# B&R Automation Studio project Agroittica
Automation Studio 4.9.5.36 SP; technology packages: mapp 5.18.0

## Configuration CP1382

CPU X20CP1382-RT, AutomationRuntime E4.83, Build 4.1.2, Safety 0.0, Vc V4.72.6

### Task classes (Cpu.sw)
```
Cyclic#1 (cycle 4000 us, tolerance 4000 us):
  Time <- main.Time.prg
  FIFO <- FIFO.FIFO.prg
  TCP_IP <- Tcp_ip.TCP_IP.prg
  Main <- main.Main.prg
  xsm_demo <- XSM_Demo_vnc.xsm_demo.prg
  xsm_demo_M <- XSM_Demo_vnc.xsm_demo_M2.prg
  Buffer_RPT <- main.Buffer_RPT.prg
  Laser_Enc <- IO.Laser_Enc.prg [disabled]
  Encoder <- IO.Encoder.prg [disabled]
Cyclic#2:
  Sim <- Sim.prg
Cyclic#3 (cycle 48000 us, tolerance 48000 us):
  RPT_CSV_ST <- main.RPT_CSV_ST.prg
Cyclic#4:
  Keys_Light <- Keys_Lights_combos.Keys_Lights.prg
  ip_adr <- XSM_Demo_vnc.ip_adr.prg  // Get ip address for VCN test.
  Recipe <- MpPkg.Recipe.prg
  Alarm_0 <- MpPkg.Alarm_0.prg
  Param_Fix <- main.Param_Fix.prg
  Hmi_Suppor <- Hmi.Hmi_Support.prg
  Login <- MpPkg.Login.prg [disabled]
DataObjects: Acp10sys
VcDataObjects: Visu_t <- Hmi.Visu_t30.dob, VGAvnc <- XSM_Demo_vnc.VGAvnc.dob, Visu <- Hmi.Visu.dob
Binaries: udbdef, arsvcreg, TCData, vcpdvnc, vcnet, vcbclass, vcrt, vcgclass, vccbtn, vcshared, vccline, vccnum, vcalarm, vccddbox, arialbd, vctcal, vcfntttf, vcdsloc, vcmgr, vccbmp, arial, vccpopup, vcpdsw, vcdsint, vcfile, vccovl, vccstr, vcctext, vccshape, vccdt, vccslider, vcchtml, vcclbox, vccscale, Visu_t01, Visu_t03, vcxml, Visu_t02, vccurl, vcpkat, vcchspot, vcpfar00, FWRules, vccalarm, Visu03, Visu01, Visu02, vcctrend, vccbar, vcpfx20, VGAvnc03, VGAvnc02, VGAvnc01, mvLoader, Acp10map, acp10cfg, ashwd, sysconf, asfw, arconfig, iomap, Recipes, AlarmHist, Alarm, ashwac, Config, Role, User, Config_1, VGAsvn01, VGAsvn03, VGAsvn02, visvc
Libraries: runtime, asstring, AsIOAcc, brsystem, AsMath, XSM_Ramp, AsIecCon, astime, Acp10_MC, sys_lib, Acp10man, Acp10par, NcGlobal, MpAlarmX, MpBase, MpRecipe, AsTCP, MpUser, MpFile, FileIO, dataobj, asarcfg, powerlnk, standard, vcresman, asbrstr, asusb, ashw, arssl, Library, visapi
```

### Hardware
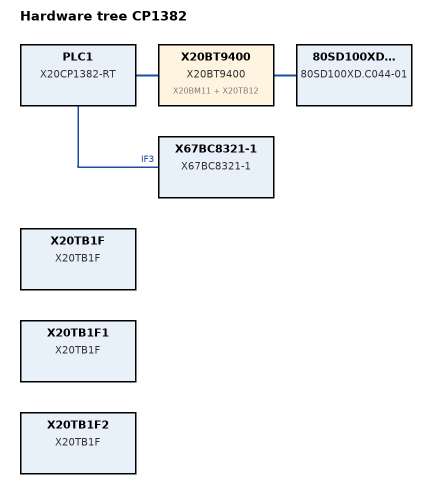
```
80SD100XD.C044-01 : 80SD100XD.C044-01 v2.2.0.0  [X2X1 -> X20BT9400.X2X1 [Cable Type=X2XCable, Length=10, Version=1.0.0.3]]
  FunctionModel = Ramp
  Supervision = off
  DirectionControl01 = on
PLC1 : X20CP1382-RT v1.11.0.0  [X1 -> X1.SL; X2 -> X2.SL; X3 -> X3.SL]
  Module X1 (Type=X1, Virtual=true, Version=1.11.0.0)
    Connection (Connector=SS1, TargetModule=X20TB1F, TargetConnector=SS)
    Connection (Connector=SL, TargetModule=PLC1, TargetConnector=X1)
    X1AI1_InputFilter = level 128
    X1AI1_InputLimitation = 4095
  Module X2 (Type=X2, Virtual=true, Version=1.11.0.0)
    Connection (Connector=SS1, TargetModule=X20TB1F1, TargetConnector=SS)
    Connection (Connector=SL, TargetModule=PLC1, TargetConnector=X2)
  Module X3 (Type=X3, Virtual=true, Version=1.11.0.0)
    Connection (Connector=SS1, TargetModule=X20TB1F2, TargetConnector=SS)
    Connection (Connector=SL, TargetModule=PLC1, TargetConnector=X3)
  Connector IF2:
    ActivateDevice = 1
    HostName = a07151
    Mode = Manual
    InternetAddress = 192.168.48.85
    SubnetMask = 255.255.255.0
    InaPort = 5555
    Vnc1
    VncVcObjectName1 = Visu_t
    VncKeyMappingFile1 = VC\PS2-Keyboard1.dis
    VncAuthentication1 = 1
    VncPasswordViewOnly1 = bazzica
    VncPasswordViewControl1 = promass
    VncMaxConnections1 = 10
    VncRefreshRate1 = 333
    Vnc2
    VncVcObjectName2 = VGAvnc
    VncKeyMappingFile2 = VC\PS2-Keyboard4.dis
    VncAuthentication2 = 1
    VncPasswordViewOnly2 = bazzica
    VncPasswordViewControl2 = promass
    VncPortNumber2 = 5901
    Vnc3
    VncVcObjectName3 = Visu
    VncKeyMappingFile3 = VC\PS2-Keyboard5.dis
    VncPortNumber3 = 5902
  Connector IF3:
    DNAConfiguration = manual
    CycleTime = 2000
    InaNodeNumber = 3
  ConfigurationID = Agroittica_CP1382
  RemanentGlobalPvSize = 100
  TimerDeviceType = EPLX2X
  TimerDevice = PLC1.IF3
  TaskClassIdleTime = 4000
  CyclicTaskClassCount = 4
  Cyclic1Duration = 4000
  Cyclic1Tolerance = 4000
  Cyclic3Duration = 48000
  Cyclic3Tolerance = 48000
  Cyclic8Duration = 8000
  FileDevice1
  FileDeviceName1 = Recipe
  FileDevicePath1 = C:\RECIPES
  FileDevice2
  FileDeviceName2 = Alarm
  FileDevicePath2 = C:\ALARM
  FileDevice3
  FileDeviceName3 = CF
  FileDevicePath3 = C:\
  FileDevice4
  FileDeviceName4 = DATA
  FileDevicePath4 = C:\DATA
  FileDevice5
  FileDeviceName5 = CFG
  FileDevicePath5 = C:\CFG
  FtpUser1
  FtpUsername1 = agroittica
  FtpUserPassword1 = lg+/2oVenYdo6VidhZ5rknSmVen51M+ANHGNxku/NAg=  // promass
  FtpUserSalt1 = EQR6eRm6
  FTPAccessRight1 = 0
  FTPdevice1 = ALL
  FtpUser2
  FtpUsername2 = bazzica
  FtpUserPassword2 = xgGZPKLqbdu5q4OkAcKaQyOUyno/5sjZu4T7S2DSwEQ=
  FtpUserSalt2 = nlL0YWjS
  FTPMSPartition2 = DATA
  ActivateOpcUa = 1
  OpcUaInformationModels_PV_Version = 1
  ReActionTaskDisabled = FALSE
X20BM11a : X20BM11 v1.0.0.1  [X2X1 -> PLC1.IF6]
X20BT9400 : X20BT9400 v1.1.0.0  [SS1 -> X20TB12a.SS; SL -> X20BM11a.SL1]
  Supervision = off
X20TB12a : X20TB12 v1.0.0.0
X20TB1F : X20TB1F v1.0.0.0
X20TB1F1 : X20TB1F v1.0.0.0
X20TB1F2 : X20TB1F v1.0.0.0
X67BC8321-1 : X67BC8321-1 v2.11.1.0  [PLK1 -> PLC1.IF3 (NodeNumber=3) [Cable Type=PowerlinkCable, Length=10, Version=1.0.0.3]]
  IOSupervision = off
  Direction01 = output
  Direction02 = output
  Direction03 = output
  Direction04 = output
  Direction05 = output
  Direction06 = output
```

### IoMap.iom - PLC1/IoMap.iom
```iecst
(********************************************************************
 * COPYRIGHT -- Bernecker + Rainer
 ********************************************************************
 * File: IoMap.iom
 * Author: leesa
 * Created: March 27, 2009
 ********************************************************************
 * IO mapping file
 ********************************************************************)
VAR_CONFIG
	::xsm_demo:XSM_Ctrl_0.IO_Mapping.ModuleOK AT %IX."80SD100XD.C044-01".ModuleOk;
	::xsm_demo:XSM_Ctrl_0.IO_Mapping.AbsPos AT %QD."80SD100XD.C044-01".AbsPos01;
	::xsm_demo:XSM_Ctrl_0.IO_Mapping.MpGenControl AT %QW."80SD100XD.C044-01".MpGenControl01;
	::xsm_demo:XSM_Ctrl_0.IO_Mapping.MpGenMode AT %QB."80SD100XD.C044-01".MpGenMode01;
	::xsm_demo:XSM_Ctrl_0.IO_Mapping.AbsPosActVal AT %ID."80SD100XD.C044-01".AbsPos01ActVal;
	::xsm_demo:XSM_Ctrl_0.IO_Mapping.MpGenStatus AT %IW."80SD100XD.C044-01".MpGenStatus01;
	::xsm_demo:XSM_Ctrl_0.IO_Mapping.InputStatus AT %IB."80SD100XD.C044-01".InputStatus;
	::xsm_demo:XSM_Ctrl_0.IO_Mapping.ModuleID AT %IW."80SD100XD.C044-01".ModuleID;
	glb_io.Di.Start AT %IX."X2".DigitalInput01;
	::xsm_demo:XSM_Ctrl_0.Enable AT %QX."X3".DigitalOutput01;
	glb_io.Do.Piston_gun_1 AT %QX."X3".DigitalOutput02;
	glb_io.Do.Piston_gun_2 AT %QX."X3".DigitalOutput04;
	Cyclic#1.Empty_Mag_22.Empty_Mag_Sensor AT %IX."X1".DigitalInput04;
	Cyclic#1.Empty_Mag_1_0.Empty_Mag_Sensor AT %IX."X1".DigitalInput02;
	::xsm_demo_M:XSM_Ctrl_2.IO_Mapping.AbsPos AT %QD."80SD100XD.C044-01".AbsPos02;
	::xsm_demo_M:XSM_Ctrl_2.IO_Mapping.MpGenControl AT %QW."80SD100XD.C044-01".MpGenControl02;
	::xsm_demo_M:XSM_Ctrl_2.IO_Mapping.MpGenMode AT %QB."80SD100XD.C044-01".MpGenMode02;
	::xsm_demo_M:XSM_Ctrl_2.IO_Mapping.AbsPosActVal AT %ID."80SD100XD.C044-01".AbsPos02ActVal;
	::xsm_demo_M:XSM_Ctrl_2.IO_Mapping.MpGenStatus AT %IW."80SD100XD.C044-01".MpGenStatus02;
	Cyclic#1.Feedback_0.Feedback_Em_Bt AT %IX."X2".DigitalInput13;
	Cyclic#1.Feedback_0.Feedback_Air AT %IX."X2".DigitalInput14;
	Cyclic#1.Beacon_1.Beeper_Alarm AT %QX."X67BC8321-1".IF1.ST1.DigitalOutput01;
	Cyclic#1.Beacon_2.Beeper_Alarm AT %QX."X67BC8321-1".IF1.ST1.DigitalOutput02;
	Cyclic#1.Beacon_1.White AT %QX."X67BC8321-1".IF1.ST1.DigitalOutput03;
	Cyclic#1.Beacon_2.White AT %QX."X67BC8321-1".IF1.ST1.DigitalOutput04;
	Cyclic#1.Beacon_1.Green AT %QX."X67BC8321-1".IF1.ST1.DigitalOutput05;
	Cyclic#1.Beacon_2.Green AT %QX."X67BC8321-1".IF1.ST1.DigitalOutput06;
	Cyclic#1.glb_io.Di.Si_03 AT %IX."X67BC8321-1".IF1.ST1.DigitalInput08;
	glb_io.Di.Powerlink AT %IX."X67BC8321-1".IF1.ST1.ModuleOk;
	glb_io.Do.Main_Piston_Up AT %QX."X3".DigitalOutput03;
	Cyclic#1.glb_io.Di.Si_01_raw AT %IX."X1".DigitalInput03;
	glb_io.Di.Automatic AT %IX."X2".DigitalInput02;
	glb_io.Di.Stop AT %IX."X2".DigitalInput03;
	glb_io.Di.Manual AT %IX."X2".DigitalInput04;
	glb_io.Di.Reset AT %IX."X2".DigitalInput05;
	glb_io.Di.Forward_Mag_1 AT %IX."X2".DigitalInput06;
	glb_io.Di.Forward_Mag_2 AT %IX."X2".DigitalInput07;
	glb_io.Di.Backward_Mag_1 AT %IX."X2".DigitalInput08;
	glb_io.Di.Backward_Mag_2 AT %IX."X2".DigitalInput09;
	glb_io.Do.Green_Light AT %QX."X3".DigitalOutput05;
	glb_io.Do.Red_Light AT %QX."X3".DigitalOutput06;
	glb_io.Do.Blue_Light AT %QX."X3".DigitalOutput07;
	glb_io.Do.Vacuum_On_Off AT %QX."X3".DigitalOutput08;
	Cyclic#1.::glb_io.Ai.Enc_laser_dist_raw AT %IW."X1".AnalogInput01;
	glb_io.Do.Main_Piston_Down AT %QX."X3".DigitalOutput09;
END_VAR
```

## Configuration CP1382_sim

### Task classes (Cpu.sw)
```
Cyclic#1 (cycle 4000 us, tolerance 4000 us):
  Sim <- Sim.prg
  Time <- main.Time.prg
  FIFO <- FIFO.FIFO.prg
  Main <- main.Main.prg
  xsm_demo <- XSM_Demo_vnc.xsm_demo.prg
  xsm_demo_M <- XSM_Demo_vnc.xsm_demo_M2.prg
  TCP_IP <- Tcp_ip.TCP_IP.prg
  Buffer_RPT <- main.Buffer_RPT.prg
  Laser_Enc <- IO.Laser_Enc.prg [disabled]
  Encoder <- IO.Encoder.prg [disabled]
Cyclic#3 (cycle 48000 us, tolerance 48000 us):
  RPT_CSV_ST <- main.RPT_CSV_ST.prg
Cyclic#4:
  Keys_Light <- Keys_Lights_combos.Keys_Lights.prg
  ip_adr <- XSM_Demo_vnc.ip_adr.prg  // Get ip address for VCN test.
  Recipe <- MpPkg.Recipe.prg
  Alarm_0 <- MpPkg.Alarm_0.prg
  Param_Fix <- main.Param_Fix.prg
  Hmi_Suppor <- Hmi.Hmi_Support.prg
  Login <- MpPkg.Login.prg [disabled]
DataObjects: Acp10sys
VcDataObjects: Visu_t <- Hmi.Visu_t30.dob, VGAvnc <- XSM_Demo_vnc.VGAvnc.dob, Visu <- Hmi.Visu.dob
Binaries: udbdef, arsvcreg, TCData, vcpdvnc, vcnet, vcbclass, vcrt, vcgclass, vccbtn, vcshared, vccline, vccnum, vcalarm, vccddbox, arialbd, vctcal, vcfntttf, vcdsloc, vcmgr, vccbmp, arial, vccpopup, vcpdsw, vcdsint, vcfile, vccovl, vccstr, vcctext, vccshape, vccdt, vccslider, vcchtml, vcclbox, vccscale, Visu_t01, Visu_t03, vcxml, Visu_t02, vccurl, vcpkat, vcchspot, vcpfar00, FWRules, vccalarm, Visu03, Visu01, Visu02, vcctrend, vccbar, VGAvnc03, VGAvnc02, VGAvnc01, mvLoader, Acp10map, acp10cfg, ashwd, sysconf, asfw, arconfig, iomap, Recipes, AlarmHist, Alarm, ashwac, Config, Role, User, Config_1, vcpfx20, VGAsvn01, VGAsvn03, VGAsvn02, visvc
ReActionTechnologyObjects: Program <- RT.Program.prg
Libraries: runtime, asstring, AsIOAcc, brsystem, AsMath, XSM_Ramp, AsIecCon, astime, Acp10_MC, sys_lib, Acp10man, Acp10par, NcGlobal, MpAlarmX, MpBase, MpRecipe, AsTCP, MpUser, MpFile, FileIO, dataobj, asarcfg, powerlnk, standard, vcresman, asbrstr, asusb, arssl, ashw, visapi, AsIORTI
```

### Hardware
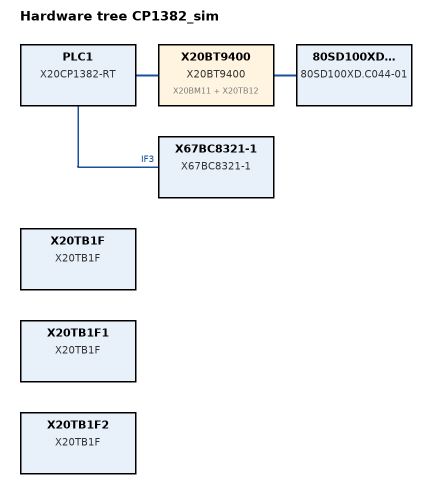
```
80SD100XD.C044-01 : 80SD100XD.C044-01 v2.2.0.0 (Disabled=true)  [X2X1 -> X20BT9400.X2X1 [Cable Type=X2XCable, Length=10, Version=1.0.0.3]]
  FunctionModel = Ramp
  Supervision = off
  DirectionControl01 = on
PLC1 : X20CP1382-RT v1.11.0.0  [X1 -> X1.SL; X2 -> X2.SL; X3 -> X3.SL]
  Module X1 (Type=X1, Virtual=true, Version=1.11.0.0)
    Connection (Connector=SS1, TargetModule=X20TB1F, TargetConnector=SS)
    Connection (Connector=SL, TargetModule=PLC1, TargetConnector=X1)
    X1AI1_InputFilter = level 128
    X1AI1_InputLimitation = 4095
  Module X2 (Type=X2, Virtual=true, Version=1.11.0.0)
    Connection (Connector=SS1, TargetModule=X20TB1F1, TargetConnector=SS)
    Connection (Connector=SL, TargetModule=PLC1, TargetConnector=X2)
  Module X3 (Type=X3, Virtual=true, Version=1.11.0.0)
    Connection (Connector=SS1, TargetModule=X20TB1F2, TargetConnector=SS)
    Connection (Connector=SL, TargetModule=PLC1, TargetConnector=X3)
  Connector IF2:
    ActivateDevice = 1
    HostName = a07151
    Mode = Manual
    InternetAddress = 192.168.48.85
    SubnetMask = 255.255.255.0
    InaPort = 5555
    Vnc1
    VncVcObjectName1 = Visu_t
    VncKeyMappingFile1 = VC\PS2-Keyboard1.dis
    VncAuthentication1 = 1
    VncPasswordViewOnly1 = bazzica
    VncPasswordViewControl1 = promass
    VncMaxConnections1 = 10
    VncRefreshRate1 = 333
    Vnc2
    VncVcObjectName2 = VGAvnc
    VncKeyMappingFile2 = VC\PS2-Keyboard4.dis
    VncAuthentication2 = 1
    VncPasswordViewOnly2 = bazzica
    VncPasswordViewControl2 = promass
    VncPortNumber2 = 5901
    Vnc3
    VncVcObjectName3 = Visu
    VncKeyMappingFile3 = VC\PS2-Keyboard5.dis
    VncPortNumber3 = 5902
  Connector IF3:
    DNAConfiguration = manual
    CycleTime = 2000
    InaNodeNumber = 3
  ConfigurationID = Agroittica_CP1382
  RemanentGlobalPvSize = 100
  TimerDeviceType = EPLX2X
  TimerDevice = PLC1.IF3
  TaskClassIdleTime = 4000
  CyclicTaskClassCount = 4
  Cyclic1Duration = 4000
  Cyclic1Tolerance = 4000
  Cyclic3Duration = 48000
  Cyclic3Tolerance = 48000
  Cyclic8Duration = 8000
  FileDevice1
  FileDeviceName1 = Recipe
  FileDevicePath1 = C:\RECIPES
  FileDevice2
  FileDeviceName2 = Alarm
  FileDevicePath2 = C:\ALARM
  FileDevice3
  FileDeviceName3 = CF
  FileDevicePath3 = C:\
  FileDevice4
  FileDeviceName4 = DATA
  FileDevicePath4 = C:\DATA
  FileDevice5
  FileDeviceName5 = CFG
  FileDevicePath5 = C:\CFG
  FtpUser1
  FtpUsername1 = agroittica
  FtpUserPassword1 = lg+/2oVenYdo6VidhZ5rknSmVen51M+ANHGNxku/NAg=  // promass
  FtpUserSalt1 = EQR6eRm6
  FTPAccessRight1 = 0
  FTPdevice1 = ALL
  FtpUser2
  FtpUsername2 = bazzica
  FtpUserPassword2 = xgGZPKLqbdu5q4OkAcKaQyOUyno/5sjZu4T7S2DSwEQ=
  FtpUserSalt2 = nlL0YWjS
  FTPMSPartition2 = DATA
  ActivateOpcUa = 1
  OpcUaInformationModels_PV_Version = 1
  ReActionTaskDisabled = FALSE
X20BM11a : X20BM11 v1.0.0.1 (Disabled=true)  [X2X1 -> PLC1.IF6]
X20BT9400 : X20BT9400 v1.1.0.0 (Disabled=true)  [SS1 -> X20TB12a.SS; SL -> X20BM11a.SL1]
  Supervision = off
X20TB12a : X20TB12 v1.0.0.0 (Disabled=true)
X20TB1F : X20TB1F v1.0.0.0
X20TB1F1 : X20TB1F v1.0.0.0
X20TB1F2 : X20TB1F v1.0.0.0
X67BC8321-1 : X67BC8321-1 v2.11.1.0 (Disabled=true)  [PLK1 -> PLC1.IF3 (NodeNumber=3) [Cable Type=PowerlinkCable, Length=10, Version=1.0.0.3]]
  Connector IF1 (Disabled=true)
  IOSupervision = off
  Direction01 = output
  Direction02 = output
  Direction03 = output
  Direction04 = output
  Direction05 = output
  Direction06 = output
```

### IoMap.iom - PLC1/IoMap.iom
```iecst
(********************************************************************
 * COPYRIGHT -- Bernecker + Rainer
 ********************************************************************
 * File: IoMap.iom
 * Author: leesa
 * Created: March 27, 2009
 ********************************************************************
 * IO mapping file
 ********************************************************************)
VAR_CONFIG
	::xsm_demo:XSM_Ctrl_0.IO_Mapping.ModuleOK AT %IX."80SD100XD.C044-01".ModuleOk;
	::xsm_demo:XSM_Ctrl_0.IO_Mapping.AbsPos AT %QD."80SD100XD.C044-01".AbsPos01;
	::xsm_demo:XSM_Ctrl_0.IO_Mapping.MpGenControl AT %QW."80SD100XD.C044-01".MpGenControl01;
	::xsm_demo:XSM_Ctrl_0.IO_Mapping.MpGenMode AT %QB."80SD100XD.C044-01".MpGenMode01;
	::xsm_demo:XSM_Ctrl_0.IO_Mapping.AbsPosActVal AT %ID."80SD100XD.C044-01".AbsPos01ActVal;
	::xsm_demo:XSM_Ctrl_0.IO_Mapping.MpGenStatus AT %IW."80SD100XD.C044-01".MpGenStatus01;
	::xsm_demo:XSM_Ctrl_0.IO_Mapping.InputStatus AT %IB."80SD100XD.C044-01".InputStatus;
	::xsm_demo:XSM_Ctrl_0.IO_Mapping.ModuleID AT %IW."80SD100XD.C044-01".ModuleID;
	glb_io.Di.Start AT %IX."X2".DigitalInput01;
	::xsm_demo:XSM_Ctrl_0.Enable AT %QX."X3".DigitalOutput01;
	glb_io.Do.Piston_gun_1 AT %QX."X3".DigitalOutput02;
	glb_io.Do.Piston_gun_2 AT %QX."X3".DigitalOutput04;
	Cyclic#1.Empty_Mag_22.Empty_Mag_Sensor AT %IX."X1".DigitalInput04;
	Cyclic#1.Empty_Mag_1_0.Empty_Mag_Sensor AT %IX."X1".DigitalInput02;
	::xsm_demo_M:XSM_Ctrl_2.IO_Mapping.AbsPos AT %QD."80SD100XD.C044-01".AbsPos02;
	::xsm_demo_M:XSM_Ctrl_2.IO_Mapping.MpGenControl AT %QW."80SD100XD.C044-01".MpGenControl02;
	::xsm_demo_M:XSM_Ctrl_2.IO_Mapping.MpGenMode AT %QB."80SD100XD.C044-01".MpGenMode02;
	::xsm_demo_M:XSM_Ctrl_2.IO_Mapping.AbsPosActVal AT %ID."80SD100XD.C044-01".AbsPos02ActVal;
	::xsm_demo_M:XSM_Ctrl_2.IO_Mapping.MpGenStatus AT %IW."80SD100XD.C044-01".MpGenStatus02;
	Cyclic#1.Feedback_0.Feedback_Em_Bt AT %IX."X2".DigitalInput13;
	Cyclic#1.Feedback_0.Feedback_Air AT %IX."X2".DigitalInput14;
	Cyclic#1.Beacon_1.Beeper_Alarm AT %QX."X67BC8321-1".IF1.ST1.DigitalOutput01;
	Cyclic#1.Beacon_2.Beeper_Alarm AT %QX."X67BC8321-1".IF1.ST1.DigitalOutput02;
	Cyclic#1.Beacon_1.White AT %QX."X67BC8321-1".IF1.ST1.DigitalOutput03;
	Cyclic#1.Beacon_2.White AT %QX."X67BC8321-1".IF1.ST1.DigitalOutput04;
	Cyclic#1.Beacon_1.Green AT %QX."X67BC8321-1".IF1.ST1.DigitalOutput05;
	Cyclic#1.Beacon_2.Green AT %QX."X67BC8321-1".IF1.ST1.DigitalOutput06;
	Cyclic#1.glb_io.Di.Si_03 AT %IX."X67BC8321-1".IF1.ST1.DigitalInput08;
	glb_io.Di.Powerlink AT %IX."X67BC8321-1".IF1.ST1.ModuleOk;
	glb_io.Do.Main_Piston_Up AT %QX."X3".DigitalOutput03;
	glb_io.Di.Si_01 AT %IX."X1".DigitalInput03;
	glb_io.Di.Automatic AT %IX."X2".DigitalInput02;
	glb_io.Di.Stop AT %IX."X2".DigitalInput03;
	glb_io.Di.Manual AT %IX."X2".DigitalInput04;
	glb_io.Di.Reset AT %IX."X2".DigitalInput05;
	glb_io.Di.Forward_Mag_1 AT %IX."X2".DigitalInput06;
	glb_io.Di.Backward_Mag_1 AT %IX."X2".DigitalInput08;
	glb_io.Di.Backward_Mag_2 AT %IX."X2".DigitalInput09;
	glb_io.Do.Green_Light AT %QX."X3".DigitalOutput05;
	glb_io.Do.Red_Light AT %QX."X3".DigitalOutput06;
	glb_io.Do.Blue_Light AT %QX."X3".DigitalOutput07;
	glb_io.Do.Vacuum_On_Off AT %QX."X3".DigitalOutput08;
	Cyclic#1.::glb_io.Ai.Enc_laser_dist_raw AT %IW."X1".AnalogInput01;
	glb_io.Do.Main_Piston_Down AT %QX."X3".DigitalOutput09;
	glb_io.Di.Forward_Mag_2 AT %IX."X2".DigitalInput07;
END_VAR
```

### Alarm.mpalarmxcore - PLC1/mappServices/Alarm.mpalarmxcore
```
Element gAlarmXCore (Type=mpalarmxcore)
  mapp.AlarmX.Core.Configuration:
    [0]:
      Name = Motor 1 fault
      Message = Motor 1 fault
      Behavior = PersistentAlarm
    [1]:
      Name = Air supply fault
      Message = Air supply not connected
      Behavior = PersistentAlarm
    [2]:
      Name = Emergency Button
      Message = Emergency Button
      Behavior = PersistentAlarm
    [3]:
      Name = Motor 2 fault
      Message = Motor 2 fault
      Behavior = PersistentAlarm
```

### Config.mpuser - PLC1/mappServices/Config.mpuser
```
Element UserMgmt (Type=mpuser)
  Groups:
    DefGroup#1:
      id = Admin
      level = 100
      admin = TRUE
      rights:
        [0] = FullAccess
        [1] = FullAccess
        [2] = FullAccess
        [3] = FullAccess
        [4] = FullAccess
    DefGroup#2:
      id = Operator
      rights:
        [0] = FullAccess
        [1] = StartOnly
        [2] = ViewOnly
        [3] = ViewOnly
        [4] = NoAccess
  Users:
    DefUser#1:
      id = Admin
      grp = Admin
      name = Default Admin User
      pwd = Admin
      pref = 
    DefUser#2:
      id = Operatore
      grp = Operator
      pwd = Agroittica
```

## Configuration CP1586

CPU X20CP1382-RT, AutomationRuntime E4.83, Build 4.1.2, Safety 0.0, Vc V4.72.6

### Task classes (Cpu.sw)
```
Cyclic#1:
  Main <- main.Main.prg
  Encoder <- IO.Encoder.prg
  xsm_demo <- XSM_Demo_vnc.xsm_demo.prg
Cyclic#4:
  ip_adr <- XSM_Demo_vnc.ip_adr.prg  // Get ip address for VCN test.
  Recipe <- MpPkg.Recipe.prg
  Alarm_0 <- MpPkg.Alarm_0.prg
  TCP_IP <- Tcp_ip.TCP_IP.prg
DataObjects: Acp10sys
VcDataObjects: VGAvnc <- XSM_Demo_vnc.VGAvnc.dob, Visu_t <- Hmi.Visu_t30.dob
Binaries: VGAvnc03, VGAvnc02, VGAvnc01, vcpdvnc, vcnet, vcbclass, vcrt, vcgclass, vccbtn, vcshared, vccline, vccnum, vcalarm, vccddbox, arialbd, vctcal, vcfntttf, vcdsloc, vcmgr, vccbmp, arial, vccpopup, vcpdsw, vcdsint, vcfile, vccovl, vccstr, vcctext, vccshape, vccdt, vccslider, vcchtml, vcclbox, vccscale, Visu_t01, Visu_t03, vcxml, Visu_t02, vccurl, vcpkat, udbdef, arsvcreg, vcchspot, TCData, vcpfx20, Acp10map, acp10cfg, ashwd, sysconf, asfw, arconfig, iomap, Recipes, AlarmHist, Alarm, ashwac, vcpfar00, VGAsvn01, VGAsvn03, VGAsvn02, visvc
Libraries: runtime, asstring, AsIOAcc, brsystem, AsMath, XSM_Ramp, AsIecCon, astime, Acp10_MC, sys_lib, Acp10man, Acp10par, NcGlobal, MpAlarmX, MpBase, MpRecipe, AsTCP, MpUser, vcresman, dataobj, asarcfg, fileio, powerlnk, standard, ashw, Library, visapi
```

### Hardware
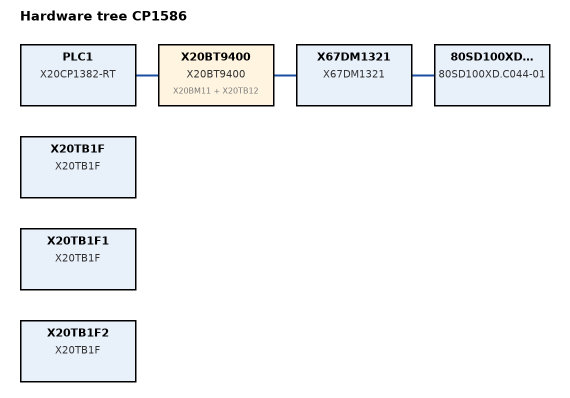
```
80SD100XD.C044-01 : 80SD100XD.C044-01 v2.2.0.0  [X2X1 -> X67DM1321.X2X2 [Cable Type=X2XCable, Length=10, Version=1.0.0.3]]
  FunctionModel = Ramp
  Supervision = off
  DirectionControl01 = on
PLC1 : X20CP1382-RT v1.11.0.0  [X1 -> X1.SL; X2 -> X2.SL; X3 -> X3.SL]
  Module X1 (Type=X1, Virtual=true, Version=1.11.0.0)
    Connection (Connector=SS1, TargetModule=X20TB1F, TargetConnector=SS)
    Connection (Connector=SL, TargetModule=PLC1, TargetConnector=X1)
  Module X2 (Type=X2, Virtual=true, Version=1.11.0.0)
    Connection (Connector=SS1, TargetModule=X20TB1F1, TargetConnector=SS)
    Connection (Connector=SL, TargetModule=PLC1, TargetConnector=X2)
  Module X3 (Type=X3, Virtual=true, Version=1.11.0.0)
    Connection (Connector=SS1, TargetModule=X20TB1F2, TargetConnector=SS)
    Connection (Connector=SL, TargetModule=PLC1, TargetConnector=X3)
    X3Channel05Config = input
    X3Channel06Config = input
    X3Channel07Config = input
    X3Channel08Config = input
    X3Channel10Source = reACTION
  Connector IF2:
    ActivateDevice = 1
    HostName = a07151
    Mode = Manual
    InternetAddress = 111.111.111.111
    SubnetMask = 255.255.255.0
    Vnc1
    VncVcObjectName1 = Visu_t
    VncKeyMappingFile1 = VC\PS2-Keyboard1.dis
    VncAuthentication1 = 1
    VncPasswordViewOnly1 = bazzica
    VncPasswordViewControl1 = promass
    VncMaxConnections1 = 10
    VncRefreshRate1 = 333
    Vnc2
    VncVcObjectName2 = VGAvnc
    VncKeyMappingFile2 = VC\PS2-Keyboard4.dis
    VncAuthentication2 = 1
    VncPasswordViewOnly2 = bazzica
    VncPasswordViewControl2 = promass
    VncPortNumber2 = 5901
  Connector IF3:
    DNAConfiguration = manual
    CycleTime = 2000
    InaNodeNumber = 1
  ConfigurationID = Agroittica_CP1382
  FileDevice1
  FileDeviceName1 = Recipe
  FileDevicePath1 = D:\RECIPES
  FileDevice2
  FileDeviceName2 = Alarm
  FileDevicePath2 = D:\ALARM
  ReActionTaskDisabled = FALSE
X20BM11a : X20BM11 v1.0.0.1  [X2X1 -> PLC1.IF6]
X20BT9400 : X20BT9400 v1.1.0.0  [SS1 -> X20TB12a.SS; SL -> X20BM11a.SL1]
  Supervision = off
X20TB12a : X20TB12 v1.0.0.0
X20TB1F : X20TB1F v1.0.0.0
X20TB1F1 : X20TB1F v1.0.0.0
X20TB1F2 : X20TB1F v1.0.0.0
X67DM1321 : X67DM1321 v1.2.0.0  [X2X1 -> X20BT9400.X2X1 [Cable Type=X2XCable, Length=10, Version=1.0.0.3]]
```

### IoMap.iom - PLC1/IoMap.iom
```iecst
(********************************************************************
 * COPYRIGHT -- Bernecker + Rainer
 ********************************************************************
 * File: IoMap.iom
 * Author: leesa
 * Created: March 27, 2009
 ********************************************************************
 * IO mapping file
 ********************************************************************)
VAR_CONFIG
	::xsm_demo:XSM_Ctrl_0.IO_Mapping.ModuleOK AT %IX."80SD100XD.C044-01".ModuleOk;
	::xsm_demo:XSM_Ctrl_0.IO_Mapping.AbsPos AT %QD."80SD100XD.C044-01".AbsPos01;
	::xsm_demo:XSM_Ctrl_0.IO_Mapping.MpGenControl AT %QW."80SD100XD.C044-01".MpGenControl01;
	::xsm_demo:XSM_Ctrl_0.IO_Mapping.MpGenMode AT %QB."80SD100XD.C044-01".MpGenMode01;
	::xsm_demo:XSM_Ctrl_0.IO_Mapping.AbsPosActVal AT %ID."80SD100XD.C044-01".AbsPos01ActVal;
	::xsm_demo:XSM_Ctrl_0.IO_Mapping.MpGenStatus AT %IW."80SD100XD.C044-01".MpGenStatus01;
	::xsm_demo:XSM_Ctrl_0.IO_Mapping.InputStatus AT %IB."80SD100XD.C044-01".InputStatus;
	::xsm_demo:XSM_Ctrl_0.IO_Mapping.ModuleID AT %IW."80SD100XD.C044-01".ModuleID;
	Cyclic#1.glb_io.Di.enc_sta_bit_00 AT %IX."X2".DigitalInput01;
	Cyclic#1.glb_io.Di.enc_sta_bit_01 AT %IX."X2".DigitalInput02;
	Cyclic#1.glb_io.Di.enc_sta_bit_02 AT %IX."X2".DigitalInput03;
	Cyclic#1.glb_io.Di.enc_sta_bit_03 AT %IX."X2".DigitalInput04;
	Cyclic#1.glb_io.Di.enc_sta_bit_04 AT %IX."X2".DigitalInput05;
	Cyclic#1.glb_io.Di.enc_sta_bit_05 AT %IX."X2".DigitalInput06;
	Cyclic#1.glb_io.Di.enc_sta_bit_06 AT %IX."X2".DigitalInput07;
	Cyclic#1.glb_io.Di.enc_sta_bit_07 AT %IX."X2".DigitalInput08;
	Cyclic#1.glb_io.Di.enc_sta_bit_08 AT %IX."X2".DigitalInput09;
	Cyclic#1.glb_io.Di.enc_sta_bit_09 AT %IX."X2".DigitalInput10;
	Cyclic#1.glb_io.Di.enc_sta_bit_10 AT %IX."X2".DigitalInput11;
	Cyclic#1.glb_io.Di.enc_sta_bit_11 AT %IX."X2".DigitalInput12;
	::xsm_demo:XSM_Ctrl_0.Enable AT %QX."X3".DigitalOutput01;
	glb_io.Di.Start AT %IX."X3".DigitalInput05;
	glb_io.Di.Automatic AT %IX."X3".DigitalInput06;
	glb_io.Di.Stop AT %IX."X3".DigitalInput07;
	glb_io.Di.Manual AT %IX."X3".DigitalInput08;
	glb_io.Do.Piston_gun_1 AT %QX."X3".DigitalOutput02;
	glb_io.Do.Piston_up AT %QX."X3".DigitalOutput03;
	glb_io.Do.Piston_gun_2 AT %QX."X3".DigitalOutput04;
	glb_io.Do.Piston_Flap_Dx_Sx AT %QX."X3".DigitalOutput09;
	Cyclic#1.Empty_Mag_22.Empty_Mag_Sensor AT %IX."X1".DigitalInput04;
	Cyclic#1.Empty_Mag_1_0.Empty_Mag_Sensor AT %IX."X1".DigitalInput02;
	::xsm_demo_M:XSM_Ctrl_2.IO_Mapping.AbsPos AT %QD."80SD100XD.C044-01".AbsPos02;
	::xsm_demo_M:XSM_Ctrl_2.IO_Mapping.MpGenControl AT %QW."80SD100XD.C044-01".MpGenControl02;
	::xsm_demo_M:XSM_Ctrl_2.IO_Mapping.MpGenMode AT %QB."80SD100XD.C044-01".MpGenMode02;
	::xsm_demo_M:XSM_Ctrl_2.IO_Mapping.AbsPosActVal AT %ID."80SD100XD.C044-01".AbsPos02ActVal;
	::xsm_demo_M:XSM_Ctrl_2.IO_Mapping.MpGenStatus AT %IW."80SD100XD.C044-01".MpGenStatus02;
	Cyclic#1.::glb_io.Di.Finecorsa AT %IX."X1".DigitalInput01;
	Cyclic#1.::glb_io.Di.Si_01 AT %IX."X1".DigitalInput03;
	Cyclic#1.Feedback_0.Feedback_PLC AT %IX."X2".DigitalInput13;
	Cyclic#1.Feedback_0.Feedback_Air AT %IX."X2".DigitalInput14;
END_VAR
```

### Alarm.mpalarmxcore - PLC1/mappServices/Alarm.mpalarmxcore
```
Element gAlarmXCore (Type=mpalarmxcore)
  mapp.AlarmX.Core.Configuration:
    [0]:
      Name = Motor 1 fault
      Message = Motor 1 fault
      Behavior = PersistentAlarm
        Retain = TRUE
    [1]:
      Name = Air supply fault
      Message = Air supply not connected
      Behavior = PersistentAlarm
        Retain = TRUE
    [2]:
      Name = Emergency Button
      Message = Emergency Button pressed
      Behavior = PersistentAlarm
        Retain = TRUE
```

## Configuration Config1

CPU X20CP1382, AutomationRuntime E4.83, Build 4.1.2, Vc V4.72.6

CPU X20CP1382-RT, AutomationRuntime E4.83, Build 4.1.2, Safety 0.0, Vc V4.72.6

### Task classes (Cpu.sw)
```
Cyclic#1:
  Main <- main.Main.prg
  Encoder <- IO.Encoder.prg
  Laser_Enc <- IO.Laser_Enc.prg
  xsm_demo <- XSM_Demo_vnc.xsm_demo.prg [disabled]
  xsm_demo_M <- XSM_Demo_vnc.xsm_demo_M2.prg [disabled]
Cyclic#4:
  Recipe <- MpPkg.Recipe.prg
  Alarm_0 <- MpPkg.Alarm_0.prg
  Login <- MpPkg.Login.prg [disabled]
VcDataObjects: Visu_t <- Hmi.Visu_t30.dob
Binaries: vcnet, udbdef, Visu_t03, vcpkat, vcctext, Visu_t01, vccurl, vcchtml, vccslider, vcfile, vcgclass, vccstr, vcpdsw, vccpopup, vccshape, arial, vccbmp, vcmgr, vctcal, vcxml, vcchspot, vcdsloc, vcfntttf, Visu_t02, vccscale, vccovl, vcshared, arialbd, vccddbox, vcalarm, vccdt, vccline, vccbtn, vcpdvnc, vcbclass, vcpfx20, vcdsint, vcrt, TCData, vcclbox, FWRules, vccnum, sysconf, iomap, Alarm, asfw, Recipes, Role, ashwac, AlarmHist, ashwd, User, arconfig
Libraries: vcresman, fileio, runtime, ashw, dataobj
```

### Task classes (Cpu.sw)
```
Cyclic#4:
  Program <- Axis.Program.prg
Libraries: McBase, MpAxis, MpBase, MpAlarmX, MpFile, MpRecipe, astime, FileIO, sys_lib, runtime
```

### Hardware
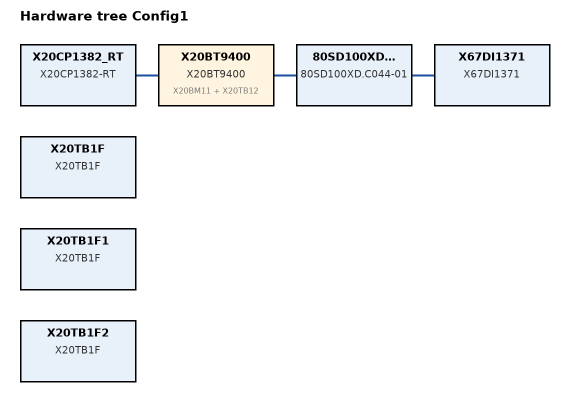
```
80SD100XD.C044-01 : 80SD100XD.C044-01 v2.2.0.0  [X2X1 -> X20BT9400.X2X1 [Cable Type=X2XCable, Length=10, Version=1.0.0.3]]
  Supervision = off
  FunctionModel/DriveConfiguration:
    ModuleParameters = StepperParameters
  FunctionModel/DriveConfiguration/ModuleParameters:
    McStepperTypeID = AcoposMicroConfig
    EncoderType = Incremental
    ReferencePulse = yes
    RatedCurrent = 10.0
    MaximumCurrent = 15.0
    AxesNumber = 2
    FullStepThreshold = 1
    StallDetection = 0
    SmartCurrentControl = 0
    BrakeOutput = 1
    NumberOfDigitalInputs = 0
    NumberOfTriggers = 2
  FunctionModel/DriveConfiguration/Channel[1]/RealAxis:
    AxisReference = gAxis_1
  FunctionModel/DriveConfiguration/Channel[1]/RealAxis/MechanicalElements/Gearbox:
    InputIsReadOnly = 0
    Input = 1
    OutputIsReadOnly = 0
    Output = 1
  FunctionModel/DriveConfiguration/Channel[1]/RealAxis/MechanicalElements/RotaryToLinearTransformation:
    ReferenceDistanceIsReadOnly = 0
    ReferenceDistance = 1
  FunctionModel/DriveConfiguration/Channel[1]/RealAxis/Motor:
    SteppingAngle = 1.8
  FunctionModel/DriveConfiguration/Channel[1]/RealAxis:
    EncoderLink = NoEncoder
  FunctionModel/DriveConfiguration/Channel[1]/RealAxis/Controller:
    ModeIsReadOnly = 0
    Mode = CurrentController
  FunctionModel/DriveConfiguration/Channel[1]/RealAxis/Controller/Mode/Current:
    StandstillCurrent = 1.1
    ConstantSpeedCurrent = 2.2
    SpeedChangeCurrent = 2.2
    FullStepThreshold = 0.0
    MotorSettlingTime = 1
    DelayedCurrentSwitchOff = 1
  FunctionModel/DriveConfiguration/Channel[1]/RealAxis/Homing:
    Mode = Direct
  FunctionModel/DriveConfiguration/Channel[1]/RealAxis/Homing/Mode:
    Position = 0.0
    ReferencePulse = NotUsed
  FunctionModel/DriveConfiguration/Channel[1]/RealAxis/Homing:
    RestorePositionVariable = 
  FunctionModel/DriveConfiguration/Channel[1]/RealAxis/StopReaction:
    DriveError = DecelerationLimit
  FunctionModel/DriveConfiguration/Channel[1]/RealAxis/MovementErrorLimits:
    PositionError = 1.0
  FunctionModel/DriveConfiguration/Channel[1]/RealAxis:
    JerkFilter = NotUsed
  FunctionModel/DriveConfiguration/Channel[1]/RealAxis/DigitalInputs/HomingSwitch:
    Source = NotUsed
    Level = High
  FunctionModel/DriveConfiguration/Channel[1]/RealAxis/DigitalInputs/PositiveLimitSwitch:
    Source = NotUsed
    Level = High
  FunctionModel/DriveConfiguration/Channel[1]/RealAxis/DigitalInputs/NegativeLimitSwitch:
    Source = NotUsed
    Level = High
  FunctionModel/DriveConfiguration/Channel[1]/RealAxis/DigitalInputs/Trigger1:
    Source = NotUsed
    Level = High
  FunctionModel/DriveConfiguration/Channel[1]/RealAxis/DigitalInputs/Trigger2:
    Source = NotUsed
    Level = High
  FunctionModel/DriveConfiguration/Channel[1]/RealAxis/DigitalInputs/Quickstop:
    Input = NotUsed
  FunctionModel/DriveConfiguration/Channel[1]/RealAxis/DigitalOutputs:
    BrakeControl = NotUsed
  FunctionModel/DriveConfiguration/Channel[2]/RealAxis:
    AxisReference = gAxis_2
  FunctionModel/DriveConfiguration/Channel[2]/RealAxis/MechanicalElements/Gearbox:
    InputIsReadOnly = 0
    Input = 1
    OutputIsReadOnly = 0
    Output = 1
  FunctionModel/DriveConfiguration/Channel[2]/RealAxis/MechanicalElements/RotaryToLinearTransformation:
    ReferenceDistanceIsReadOnly = 0
    ReferenceDistance = 1
  FunctionModel/DriveConfiguration/Channel[2]/RealAxis/Motor:
    SteppingAngle = 1.8
  FunctionModel/DriveConfiguration/Channel[2]/RealAxis:
    EncoderLink = NoEncoder
  FunctionModel/DriveConfiguration/Channel[2]/RealAxis/Controller:
    ModeIsReadOnly = 0
    Mode = CurrentController
  FunctionModel/DriveConfiguration/Channel[2]/RealAxis/Controller/Mode/Current:
    StandstillCurrent = 0.3
    ConstantSpeedCurrent = 1.5
    SpeedChangeCurrent = 3
    FullStepThreshold = 0.0
    MotorSettlingTime = 1
    DelayedCurrentSwitchOff = 1
  FunctionModel/DriveConfiguration/Channel[2]/RealAxis/Homing:
    Mode = Direct
  FunctionModel/DriveConfiguration/Channel[2]/RealAxis/Homing/Mode:
    Position = 0.0
    ReferencePulse = NotUsed
  FunctionModel/DriveConfiguration/Channel[2]/RealAxis/Homing:
    RestorePositionVariable = 
  FunctionModel/DriveConfiguration/Channel[2]/RealAxis/StopReaction:
    DriveError = DecelerationLimit
  FunctionModel/DriveConfiguration/Channel[2]/RealAxis/MovementErrorLimits:
    PositionError = 1.0
  FunctionModel/DriveConfiguration/Channel[2]/RealAxis:
    JerkFilter = NotUsed
  FunctionModel/DriveConfiguration/Channel[2]/RealAxis/DigitalInputs/HomingSwitch:
    Source = NotUsed
    Level = High
  FunctionModel/DriveConfiguration/Channel[2]/RealAxis/DigitalInputs/PositiveLimitSwitch:
    Source = NotUsed
    Level = High
  FunctionModel/DriveConfiguration/Channel[2]/RealAxis/DigitalInputs/NegativeLimitSwitch:
    Source = NotUsed
    Level = High
  FunctionModel/DriveConfiguration/Channel[2]/RealAxis/DigitalInputs/Trigger1:
    Source = NotUsed
    Level = High
  FunctionModel/DriveConfiguration/Channel[2]/RealAxis/DigitalInputs/Trigger2:
    Source = NotUsed
    Level = High
  FunctionModel/DriveConfiguration/Channel[2]/RealAxis/DigitalInputs/Quickstop:
    Input = NotUsed
  FunctionModel/DriveConfiguration/Channel[2]/RealAxis/DigitalOutputs:
    BrakeControl = NotUsed
X20BM11 : X20BM11 v1.0.0.1  [X2X1 -> X20CP1382_RT.IF6]
X20BT9400 : X20BT9400 v1.1.0.0  [SS1 -> X20TB12.SS; SL -> X20BM11.SL1]
  Supervision = off
X20CP1382_RT : X20CP1382-RT v1.11.0.0  [X1 -> X1.SL; X2 -> X2.SL; X3 -> X3.SL]
  Module X1 (Type=X1, Virtual=true, Version=1.11.0.0)
    Connection (Connector=SS1, TargetModule=X20TB1F, TargetConnector=SS)
    Connection (Connector=SL, TargetModule=X20CP1382_RT, TargetConnector=X1)
  Module X2 (Type=X2, Virtual=true, Version=1.11.0.0)
    Connection (Connector=SS1, TargetModule=X20TB1F1, TargetConnector=SS)
    Connection (Connector=SL, TargetModule=X20CP1382_RT, TargetConnector=X2)
  Module X3 (Type=X3, Virtual=true, Version=1.11.0.0)
    Connection (Connector=SS1, TargetModule=X20TB1F2, TargetConnector=SS)
    Connection (Connector=SL, TargetModule=X20CP1382_RT, TargetConnector=X3)
  Connector IF2:
    ActivateDevice = 1
    Mode = Manual
    InternetAddress = 192.168.250.100
    SubnetMask = 255.255.255.0
    InaNodeNumber = 0
    ActivateModbus = 1
    NumSlaves = -1
    NumAllBlocks = -1
    MemSizeIn = -1
    MemSizeOut = -1
    ModbusSlaveGrey = 1
    ModbusSlaveConfig_1
    HoldingRegisterChannelGroup1_1
    HoldingRegisterChannelID1_1 = Statusword_6041
    HoldingRegisterChannelAddress1_1 = 6041
    HoldingRegisterChannelType1_1 = UINT
  ConfigurationID = Agroittica_Config1
  ReActionTaskDisabled = FALSE
X20TB12 : X20TB12 v1.0.0.0
X20TB1F : X20TB1F v1.0.0.0
X20TB1F1 : X20TB1F v1.0.0.0
X20TB1F2 : X20TB1F v1.0.0.0
X67DI1371 : X67DI1371 v1.1.0.0 (Disabled=true)  [X2X1 -> 80SD100XD.C044-01.X2X2 [Cable Type=X2XCable, Length=10, Version=1.0.0.3]]
  Supervision = off
```

### IoMap.iom - X20CP1382/IoMap.iom
```iecst
VAR_CONFIG
	Cyclic#3.glb_io.Ai.Enc_laser_dist_raw AT %IW."X1a".AnalogInput01;
	glb_io.Ai.Enc_laser_dist_raw1 AT %IW."X20AI4632".AnalogInput01;
	glb_io.Do.Main_Piston_Up AT %QX."X3a".DigitalOutput01;
	glb_io.Di.Si_01 AT %IX."X2a".DigitalInput01;
END_VAR
```

## Configuration Cp1301

CPU X20CP1301, AutomationRuntime C4.73, Build 4.1.2, Vc V4.72.6

### Task classes (Cpu.sw)
```
Cyclic#1 (cycle 40000 us, tolerance 40000 us):
  FIFO <- FIFO.FIFO.prg
  Main <- main.Main.prg
  Buffer_RPT <- main.Buffer_RPT.prg
  Time <- main.Time.prg
  Encoder <- IO.Encoder.prg
  TCP_IP <- Tcp_ip.TCP_IP.prg
Cyclic#2:
  Sim <- Sim.prg
Cyclic#3:
  RPT_CSV_ST <- main.RPT_CSV_ST.prg
  ip_adr <- XSM_Demo_vnc.ip_adr.prg
Cyclic#5:
  Param_Fix <- main.Param_Fix.prg
  Hmi_Suppor <- Hmi.Hmi_Support.prg
VcDataObjects: Visu_t <- Hmi.Visu_t30.dob
Binaries: vcctext, arialbd, vcmgr, vccpopup, vcxml, vccdt, vccshape, vcpkat, vcchspot, vcnet, vcdsloc, vcbclass, vcfntttf, vccovl, vcdsint, Visu_t01, vctcal, Visu_t03, vcshared, vcrt, vcpdsw, vccbmp, TCData, vcfile, vccbtn, vccslider, vccddbox, vcalarm, vccnum, FWRules, arial, Visu_t02, udbdef, vccscale, vccline, vcpdvnc, vccstr, vcchtml, vcctrend, vcgclass, vcclbox, vccurl, vcpfx20, Role, arconfig, User, asfw, ashwd, ashwac, sysconf, iomap
Libraries: asieccon, ashw, dataobj, asmath, vcresman, asarcfg, runtime, astime, standard, asstring, fileio, astcp
```

### Hardware
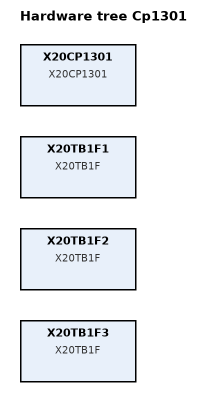
```
X20CP1301 : X20CP1301 v1.7.0.0  [X1 -> X1a.SL; X2 -> X2a.SL; X3 -> X3a.SL]
  Module X1a (Type=X1, Virtual=true, Version=1.7.0.0)
    Connection (Connector=SS1, TargetModule=X20TB1F1, TargetConnector=SS)
    Connection (Connector=SL, TargetModule=X20CP1301, TargetConnector=X1)
  Module X2a (Type=X2, Virtual=true, Version=1.7.0.0)
    Connection (Connector=SS1, TargetModule=X20TB1F2, TargetConnector=SS)
    Connection (Connector=SL, TargetModule=X20CP1301, TargetConnector=X2)
  Module X3a (Type=X3, Virtual=true, Version=1.7.0.0)
    Connection (Connector=SS1, TargetModule=X20TB1F3, TargetConnector=SS)
    Connection (Connector=SL, TargetModule=X20CP1301, TargetConnector=X3)
  Connector IF2:
    ActivateDevice = 1
    Mode = Manual
    InternetAddress = 192.168.32.200
    SubnetMask = 255.255.255.0
    Vnc1
    VncVcObjectName1 = Visu_t
    VncKeyMappingFile1 = VC\PS2-Keyboard.dis
    VncMaxConnections1 = 5
  ConfigurationID = Agroittica_Cp1301
  RemanentGlobalPvSize = 5000
  TimerDeviceType = EPLX2X
  TimerDevice = X20CP1301.IF6
  CyclicTaskClassCount = 5
  Cyclic1Duration = 40000
  Cyclic1Tolerance = 40000
  FileDevice1
  FileDeviceName1 = CF
  FileDevicePath1 = C:\
  FileDevice2
  FileDeviceName2 = DATA
  FileDevicePath2 = C:\DATA
  FtpUser1
  FtpUsername1 = promass
  FtpUserPassword1 = zPi2wKmuH/Kd7eFrewHi5384RVXQKBIyEFEQ8dCJ90M=
  FtpUserSalt1 = L1XkAkhN
  FTPAccessRight1 = 0
  FTPdevice1 = ALL
X20TB1F1 : X20TB1F v1.0.0.0
X20TB1F2 : X20TB1F v1.0.0.0
X20TB1F3 : X20TB1F v1.0.0.0
```

## Configuration Simulazione

### Task classes (Cpu.sw)
```
Cyclic#1:
  Sim <- Sim.prg
  Allarm <- Allarmi.Allarm.prg [disabled]
  xsm_demo_M <- XSM_Demo_vnc.xsm_demo_M2.prg
  Main <- main.Main.prg
  Encoder <- IO.Encoder.prg
  xsm_demo <- XSM_Demo_vnc.xsm_demo.prg
Cyclic#4:
  ip_adr <- XSM_Demo_vnc.ip_adr.prg  // Get ip address for VCN test.
  Recipe <- MpPkg.Recipe.prg
  Alarm_0 <- MpPkg.Alarm_0.prg
  TCP_IP <- Tcp_ip.TCP_IP.prg
  Login <- MpPkg.Login.prg [disabled]
DataObjects: Acp10sys
VcDataObjects: Visu_t <- main.Main.Hmi.Visu_t30.dob, VGAvnc <- XSM_Demo_vnc.VGAvnc.dob [disabled]
Binaries: udbdef, arsvcreg, TCData, vcpdvnc, vcnet, vcbclass, vcrt, vcgclass, vccbtn, vcshared, vccline, vccnum, vcalarm, vccddbox, arialbd, vctcal, vcfntttf, vcdsloc, vcmgr, vccbmp, arial, vccpopup, vcpdsw, vcdsint, vcfile, vccovl, vccstr, vcctext, vccshape, vccdt, vccslider, vcchtml, vcclbox, vccscale, Visu_t01, Visu_t03, vcxml, Visu_t02, vccurl, vcpkat, vcchspot, vcpfar00, Acp10map, acp10cfg, ashwd, sysconf, asfw, arconfig, iomap, Recipes, AlarmHist, Alarm, ashwac, vcpfx20, VGAvnc03, VGAvnc02, VGAvnc01, VGAsvn01, VGAsvn03, VGAsvn02, visvc
Libraries: runtime, asstring, AsIOAcc, brsystem, AsMath, XSM_Ramp, AsIecCon, astime, Acp10_MC, sys_lib, Acp10man, Acp10par, NcGlobal, MpAlarmX, MpBase, MpRecipe, AsTCP, MpUser, MpFile, FileIO, dataobj, asarcfg, powerlnk, standard, vcresman, asbrstr, asusb, ashw, Library, visapi
```

### Hardware
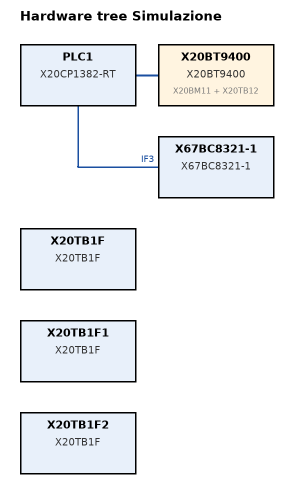
```
PLC1 : X20CP1382-RT v1.11.0.0  [X1 -> X1.SL; X2 -> X2.SL; X3 -> X3.SL]
  Module X1 (Type=X1, Virtual=true, Version=1.11.0.0)
    Connection (Connector=SS1, TargetModule=X20TB1F, TargetConnector=SS)
    Connection (Connector=SL, TargetModule=PLC1, TargetConnector=X1)
  Module X2 (Type=X2, Virtual=true, Version=1.11.0.0)
    Connection (Connector=SS1, TargetModule=X20TB1F1, TargetConnector=SS)
    Connection (Connector=SL, TargetModule=PLC1, TargetConnector=X2)
  Module X3 (Type=X3, Virtual=true, Version=1.11.0.0)
    Connection (Connector=SS1, TargetModule=X20TB1F2, TargetConnector=SS)
    Connection (Connector=SL, TargetModule=PLC1, TargetConnector=X3)
    X3Channel05Config = input
    X3Channel06Config = input
    X3Channel07Config = input
    X3Channel08Config = input
  Connector IF2:
    ActivateDevice = 1
    HostName = a07151
    Mode = Manual
    InternetAddress = 111.111.111.111
    SubnetMask = 255.255.255.0
    Vnc1
    VncVcObjectName1 = Visu_t
    VncKeyMappingFile1 = VC\PS2-Keyboard1.dis
    VncAuthentication1 = 1
    VncPasswordViewOnly1 = bazzica
    VncPasswordViewControl1 = promass
    VncMaxConnections1 = 10
    VncRefreshRate1 = 333
    Vnc2
    VncVcObjectName2 = VGAvnc
    VncKeyMappingFile2 = VC\PS2-Keyboard4.dis
    VncAuthentication2 = 1
    VncPasswordViewOnly2 = bazzica
    VncPasswordViewControl2 = promass
    VncPortNumber2 = 5901
  Connector IF3:
    DNAConfiguration = manual
    CycleTime = 2000
    InaNodeNumber = 3
  ConfigurationID = Agroittica_CP1382
  Simulation = 1
  FileDevice1
  FileDeviceName1 = Recipe
  FileDevicePath1 = D:\RECIPES
  FileDevice2
  FileDeviceName2 = Alarm
  FileDevicePath2 = D:\ALARM
  ReActionTaskDisabled = FALSE
X20BM11a : X20BM11 v1.0.0.1  [X2X1 -> PLC1.IF6]
X20BT9400 : X20BT9400 v1.1.0.0  [SS1 -> X20TB12a.SS; SL -> X20BM11a.SL1]
  Supervision = off
X20TB12a : X20TB12 v1.0.0.0
X20TB1F : X20TB1F v1.0.0.0
X20TB1F1 : X20TB1F v1.0.0.0
X20TB1F2 : X20TB1F v1.0.0.0
X67BC8321-1 : X67BC8321-1 v2.11.1.0  [PLK1 -> PLC1.IF3 (NodeNumber=3) [Cable Type=PowerlinkCable, Length=10, Version=1.0.0.3]]
  IOSupervision = off
  Direction01 = output
  Direction02 = output
  Direction03 = output
  Direction04 = output
  Direction05 = output
  Direction06 = output
```

### IoMap.iom - PLC1/IoMap.iom
```iecst
(********************************************************************
 * COPYRIGHT -- Bernecker + Rainer
 ********************************************************************
 * File: IoMap.iom
 * Author: leesa
 * Created: March 27, 2009
 ********************************************************************
 * IO mapping file
 ********************************************************************)
VAR_CONFIG
	Cyclic#1.Lamp_02.Lamp2Allarme AT %QX."X67BC8321-1".IF1.ST1.DigitalOutput01;
	Cyclic#1.Lamp_01.Lamp1Allarme AT %QX."X67BC8321-1".IF1.ST1.DigitalOutput02;
	Cyclic#1.Lamp_02.Lamp2Bianco AT %QX."X67BC8321-1".IF1.ST1.DigitalOutput03;
	Cyclic#1.Lamp_01.Lamp1Bianco AT %QX."X67BC8321-1".IF1.ST1.DigitalOutput04;
	Cyclic#1.Lamp_02.Lamp2Verde AT %QX."X67BC8321-1".IF1.ST1.DigitalOutput05;
	Cyclic#1.Lamp_01.Lamp1Verde AT %QX."X67BC8321-1".IF1.ST1.DigitalOutput06;
END_VAR
```

## Configuration Test_Mapp_View

CPU X20CP1382-RT, AutomationRuntime E4.83, Build 4.1.2, Safety 0.0, Vc V4.72.6

### Acp10cfg.ncc - PLC1/Motion/Acp10cfg.ncc
```
NcConfiguration (Version=5.22.1, NcSwId=Acp10)
  ACP10CF1_typ:
    cnt_nettrc_rec_drive = 150
    bufsize_trace_upload = 1200
    tc_nc_man_task = Cyclic #1
    glob_pv_as_ncobject = Yes
    ncsys_dl_broadcast = Yes
    ncsys_dl_acp_reset = Yes
    safemc_log_err_to_ax = Yes
    network_init:
      ncsw_init_execute = Yes
      automatic_execute = No
      node_nr_warning = Yes
      net_err_before_ncact = Yes
    nettrc:
      enter_parsecrec = Yes
      enter_ncaction = Yes
      save_ring_startidx = No
    cam_prof_download:
      cam_dat_dl_parallel = No
      tc_cam_dl_parallel = Task class for NC Manager task
```

### Config_1.mpuserlogin - PLC1/mappServices/Config_1.mpuserlogin
```
Element gUserLogin (Type=mpuserlogin)
```

## Configuration Test_Vision

CPU X20CP1382-RT, AutomationRuntime E4.83, Build 4.1.2, Safety 0.0, Vc V4.72.6

### Task classes (Cpu.sw)
```
Cyclic#1:
  Time <- main.Time.prg
  FIFO <- FIFO.FIFO.prg
  Main <- main.Main.prg
  xsm_demo <- XSM_Demo_vnc.xsm_demo.prg
  xsm_demo_M <- XSM_Demo_vnc.xsm_demo_M2.prg
  TCP_IP <- Tcp_ip.TCP_IP.prg
  Buffer_RPT <- main.Buffer_RPT.prg
  Laser_Enc <- IO.Laser_Enc.prg [disabled]
  Encoder <- IO.Encoder.prg [disabled]
Cyclic#2:
  Sim <- Sim.prg
Cyclic#3:
  RPT_CSV_ST <- main.RPT_CSV_ST.prg
Cyclic#4:
  Keys_Light <- Keys_Lights_combos.Keys_Lights.prg
  ip_adr <- XSM_Demo_vnc.ip_adr.prg  // Get ip address for VCN test.
  Recipe <- MpPkg.Recipe.prg
  Alarm_0 <- MpPkg.Alarm_0.prg
  Param_Fix <- main.Param_Fix.prg
  Hmi_Suppor <- Hmi.Hmi_Support.prg
  Login <- MpPkg.Login.prg [disabled]
DataObjects: Acp10sys
VcDataObjects: Visu_t <- Hmi.Visu_t30.dob, VGAvnc <- XSM_Demo_vnc.VGAvnc.dob, Visu <- Hmi.Visu.dob
Binaries: udbdef, arsvcreg, TCData, vcpdvnc, vcnet, vcbclass, vcrt, vcgclass, vccbtn, vcshared, vccline, vccnum, vcalarm, vccddbox, arialbd, vctcal, vcfntttf, vcdsloc, vcmgr, vccbmp, arial, vccpopup, vcpdsw, vcdsint, vcfile, vccovl, vccstr, vcctext, vccshape, vccdt, vccslider, vcchtml, vcclbox, vccscale, Visu_t01, Visu_t03, vcxml, Visu_t02, vccurl, vcpkat, vcchspot, vcpfar00, FWRules, vccalarm, Visu03, Visu01, Visu02, vcctrend, vccbar, vcpfx20, VGAvnc03, VGAvnc02, VGAvnc01, Acp10map, acp10cfg, ashwd, sysconf, asfw, arconfig, iomap, Recipes, AlarmHist, Alarm, ashwac, Config, Role, User, Config_1, VGAsvn01, VGAsvn03, VGAsvn02, visvc
Libraries: runtime, asstring, AsIOAcc, brsystem, AsMath, XSM_Ramp, AsIecCon, astime, Acp10_MC, sys_lib, Acp10man, Acp10par, NcGlobal, MpAlarmX, MpBase, MpRecipe, AsTCP, MpUser, MpFile, FileIO, dataobj, asarcfg, powerlnk, standard, vcresman, asbrstr, asusb, ashw, Library, visapi
```

### IoMap.iom - PLC1/IoMap.iom
```iecst
(********************************************************************
 * COPYRIGHT -- Bernecker + Rainer
 ********************************************************************
 * File: IoMap.iom
 * Author: leesa
 * Created: March 27, 2009
 ********************************************************************
 * IO mapping file
 ********************************************************************)
VAR_CONFIG
	::xsm_demo:XSM_Ctrl_0.IO_Mapping.ModuleOK AT %IX."80SD100XD.C044-01".ModuleOk;
	::xsm_demo:XSM_Ctrl_0.IO_Mapping.AbsPos AT %QD."80SD100XD.C044-01".AbsPos01;
	::xsm_demo:XSM_Ctrl_0.IO_Mapping.MpGenControl AT %QW."80SD100XD.C044-01".MpGenControl01;
	::xsm_demo:XSM_Ctrl_0.IO_Mapping.MpGenMode AT %QB."80SD100XD.C044-01".MpGenMode01;
	::xsm_demo:XSM_Ctrl_0.IO_Mapping.AbsPosActVal AT %ID."80SD100XD.C044-01".AbsPos01ActVal;
	::xsm_demo:XSM_Ctrl_0.IO_Mapping.MpGenStatus AT %IW."80SD100XD.C044-01".MpGenStatus01;
	::xsm_demo:XSM_Ctrl_0.IO_Mapping.InputStatus AT %IB."80SD100XD.C044-01".InputStatus;
	::xsm_demo:XSM_Ctrl_0.IO_Mapping.ModuleID AT %IW."80SD100XD.C044-01".ModuleID;
	glb_io.Di.Start AT %IX."X2".DigitalInput01;
	::xsm_demo:XSM_Ctrl_0.Enable AT %QX."X3".DigitalOutput01;
	glb_io.Do.Piston_gun_1 AT %QX."X3".DigitalOutput02;
	glb_io.Do.Piston_gun_2 AT %QX."X3".DigitalOutput04;
	Cyclic#1.Empty_Mag_22.Empty_Mag_Sensor AT %IX."X1".DigitalInput04;
	Cyclic#1.Empty_Mag_1_0.Empty_Mag_Sensor AT %IX."X1".DigitalInput02;
	::xsm_demo_M:XSM_Ctrl_2.IO_Mapping.AbsPos AT %QD."80SD100XD.C044-01".AbsPos02;
	::xsm_demo_M:XSM_Ctrl_2.IO_Mapping.MpGenControl AT %QW."80SD100XD.C044-01".MpGenControl02;
	::xsm_demo_M:XSM_Ctrl_2.IO_Mapping.MpGenMode AT %QB."80SD100XD.C044-01".MpGenMode02;
	::xsm_demo_M:XSM_Ctrl_2.IO_Mapping.AbsPosActVal AT %ID."80SD100XD.C044-01".AbsPos02ActVal;
	::xsm_demo_M:XSM_Ctrl_2.IO_Mapping.MpGenStatus AT %IW."80SD100XD.C044-01".MpGenStatus02;
	Cyclic#1.Feedback_0.Feedback_Em_Bt AT %IX."X2".DigitalInput13;
	Cyclic#1.Feedback_0.Feedback_Air AT %IX."X2".DigitalInput14;
	Cyclic#1.Beacon_1.Beeper_Alarm AT %QX."X67BC8321-1".IF1.ST1.DigitalOutput01;
	Cyclic#1.Beacon_2.Beeper_Alarm AT %QX."X67BC8321-1".IF1.ST1.DigitalOutput02;
	Cyclic#1.Beacon_1.White AT %QX."X67BC8321-1".IF1.ST1.DigitalOutput03;
	Cyclic#1.Beacon_2.White AT %QX."X67BC8321-1".IF1.ST1.DigitalOutput04;
	Cyclic#1.Beacon_1.Green AT %QX."X67BC8321-1".IF1.ST1.DigitalOutput05;
	Cyclic#1.Beacon_2.Green AT %QX."X67BC8321-1".IF1.ST1.DigitalOutput06;
	Cyclic#1.glb_io.Di.Si_03 AT %IX."X67BC8321-1".IF1.ST1.DigitalInput08;
	glb_io.Di.Powerlink AT %IX."X67BC8321-1".IF1.ST1.ModuleOk;
	Cyclic#1.::glb_io.Ai.Enc_laser_dist_raw AT %IW."X1".AnalogInput01;
	glb_io.Do.Main_Piston_Down AT %QX."X3".DigitalOutput10;
	glb_io.Do.Main_Piston_Up AT %QX."X3".DigitalOutput03;
	glb_io.Di.Si_01 AT %IX."X1".DigitalInput03;
	glb_io.Di.Automatic AT %IX."X2".DigitalInput02;
	glb_io.Di.Stop AT %IX."X2".DigitalInput03;
	glb_io.Di.Manual AT %IX."X2".DigitalInput04;
	glb_io.Di.Reset AT %IX."X2".DigitalInput05;
	glb_io.Di.Forward_Mag_1 AT %IX."X2".DigitalInput06;
	glb_io.Di.Forward_Mag_2 AT %IX."X2".DigitalInput07;
	glb_io.Di.Backward_Mag_1 AT %IX."X2".DigitalInput08;
	glb_io.Di.Backward_Mag_2 AT %IX."X2".DigitalInput09;
	glb_io.Do.Green_Light AT %QX."X3".DigitalOutput05;
	glb_io.Do.Red_Light AT %QX."X3".DigitalOutput06;
	glb_io.Do.Blue_Light AT %QX."X3".DigitalOutput07;
	glb_io.Do.Vacuum_On_Off AT %QX."X3".DigitalOutput08;
END_VAR
```

## Configuration ppc2100

CPU 5PPC2100.BY34-000, AutomationRuntime E4.83, Build 4.1.2, Safety 0.0, Vc V4.72.6

### Task classes (Cpu.sw)
```
Cyclic#4:
  io_drive <- IO.io_drive.prg
  TCP_IP <- Tcp_ip.TCP_IP.prg
  Main <- main.Main.prg
  Recipe <- MpPkg.Recipe.prg
  Alarm_0 <- MpPkg.Alarm_0.prg
VcDataObjects: Visu <- Hmi.Visu.dob, Visu_T <- Hmi.Visu_T30.dob
Libraries: AsTCP, runtime, standard, asstring, MpRecipe, MpBase, sys_lib, MpFile, FileIO, MpAlarmX, astime
```

### Hardware
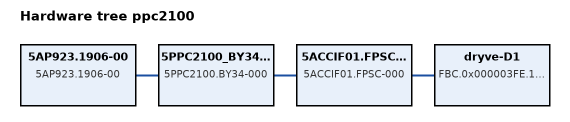
```
5ACCIF01.FPSC-000 : 5ACCIF01.FPSC-000 v1.9.2.0  [SL -> 5PPC2100_BY34_000.SL1]
  Connector IF3:
    ActivateCanOpen = 1
    pnmtstartup_maximumbootuptime = 60
    procPriority = 197
5AP923.1906-00 : 5AP923.1906-00 v2.0.0.0
  VcObjectName = Visu
5PPC2100_BY34_000 : 5PPC2100.BY34-000 v2.1.0.0  [SY -> 5AP923.1906-00.SY1]
  Connector IF3:
    AssignedOperatingSystem = ARemb
    ActivateDevice = 1
    Mode = Manual
    InternetAddress = 192.168.250.90
    SubnetMask = 255.255.255.0
    Vnc1
    VncVcObjectName1 = Visu
    VncKeyMappingFile1 = VC\PS2-Keyboard.dis
    VncAuthentication1 = 1
    VncPasswordViewOnly1 = bazzica
    VncPasswordViewControl1 = promass
    VncMaxConnections1 = 3
    Vnc2
    VncVcObjectName2 = Visu_T
    VncKeyMappingFile2 = VC\PS2-Keyboard1.dis
    VncAuthentication2 = 1
    VncPasswordViewOnly2 = bazzica
    VncPasswordViewControl2 = promass
    VncPortNumber2 = 5901
    VncMaxConnections2 = 3
  Connector IF4:
    AssignedOperatingSystem = ARemb
    ActivateDevice = 1
  Connector IF5:
    AssignedOperatingSystem = ARemb
  Connector IF6:
    AssignedOperatingSystem = ARemb
  ConfigurationID = Agroittica_ppc2100
  FileDevice1
  FileDeviceName1 = Recipe
  FileDevicePath1 = d:\RECIPES\
  FileDevice2
  FileDeviceName2 = Alarm
  FileDevicePath2 = d:\ALARM\
  FtpUser1
  FtpUsername1 = bazzica
  FtpUserPassword1 = Ug7+o3w42OmJA3hz7c8pCplDp9FITZ+DMLVGo1h2j0Y=
  FtpUserSalt1 = /4pfi4m9
  FTPAccessRight1 = 0
  FTPMSPartition1 = DATA
dryve-D1 : FBC.0x000003FE.1.20220118-dryve-D1-8PDO v1.13 (OrderNumber=dryve-D1)  [CAN1 -> 5ACCIF01.FPSC-000.IF3 (NodeNumber=2)]
  p603f_connecttomaster = 1
  p6060_connecttomaster = 3
  p6061_connecttomaster = 3
  p607f_connecttomaster = 7
  p607f_parametervalue = 0x5
  p6081_connecttomaster = 4
  p6083_connecttomaster = 4
  p6092sub1_connecttomaster = 1
  p6092sub2_connecttomaster = 5
  p6099sub1_connecttomaster = 6
  p6099sub2_connecttomaster = 5
  p609a_connecttomaster = 6
  p60c5_connecttomaster = 2
  pheartbeat_producertime = 500
  p1003_objflags = 1
  p1003sub0_objflags = 1
  p1005_objflags = 1
  p1006_objflags = 1
  p1007_objflags = 1
  p1008_objflags = 1
  p1009_objflags = 1
  p100a_objflags = 1
  p1010_objflags = 1
  p1010sub0_objflags = 1
  p1010sub1_objflags = 1
  p1010sub2_objflags = 1
  p1010sub3_objflags = 1
  p1014_objflags = 1
  p1015_objflags = 1
  p1018_objflags = 1
  p1018sub0_objflags = 1
  p1200_objflags = 1
  p1200sub0_objflags = 1
  p1200sub1_objflags = 1
  p2000 (Disabled=true)
  p2000_parametername =  (Disabled=true)
  p2000_objecttype =  (Disabled=true)
  p2000_datatype =  (Disabled=true)
  p2000_subnumber =  (Disabled=true)
  p2000_parametervalue =  (Disabled=true)
  p2000_objflags = 1 (Disabled=true)
  p2000sub0 (Disabled=true)
  p2000sub0_parametername =  (Disabled=true)
  p2000sub0_objecttype =  (Disabled=true)
  p2000sub0_datatype =  (Disabled=true)
  p2000sub0_accesstype =  (Disabled=true)
  p2000sub0_pdomapping =  (Disabled=true)
  p2000sub0_parametervalue =  (Disabled=true)
  p2000sub0_objflags = 1 (Disabled=true)
  p2000sub2 (Disabled=true)
  p2000sub2_parametername =  (Disabled=true)
  p2000sub2_objecttype =  (Disabled=true)
  p2000sub2_datatype =  (Disabled=true)
  p2000sub2_accesstype =  (Disabled=true)
  p2000sub2_pdomapping =  (Disabled=true)
  p2000sub2_parametervalue =  (Disabled=true)
  p2000sub2_objflags = 1 (Disabled=true)
  p2000sub3 (Disabled=true)
  p2000sub3_parametername =  (Disabled=true)
  p2000sub3_objecttype =  (Disabled=true)
  p2000sub3_datatype =  (Disabled=true)
  p2000sub3_accesstype =  (Disabled=true)
  p2000sub3_pdomapping =  (Disabled=true)
  p2000sub3_parametervalue =  (Disabled=true)
  p2000sub3_objflags = 1 (Disabled=true)
  p2001 (Disabled=true)
  p2001_parametername =  (Disabled=true)
  p2001_objecttype =  (Disabled=true)
  p2001_datatype =  (Disabled=true)
  p2001_accesstype =  (Disabled=true)
  p2001_pdomapping =  (Disabled=true)
  p2001_parametervalue =  (Disabled=true)
  p2001_objflags = 1 (Disabled=true)
  p2002 (Disabled=true)
  p2002_parametername =  (Disabled=true)
  p2002_objecttype =  (Disabled=true)
  p2002_datatype =  (Disabled=true)
  p2002_accesstype =  (Disabled=true)
  p2002_pdomapping =  (Disabled=true)
  p2002_parametervalue =  (Disabled=true)
  p2002_objflags = 1 (Disabled=true)
  p2003 (Disabled=true)
  p2003_parametername =  (Disabled=true)
  p2003_objecttype =  (Disabled=true)
  p2003_datatype =  (Disabled=true)
  p2003_subnumber =  (Disabled=true)
  p2003_parametervalue =  (Disabled=true)
  p2003_objflags = 1 (Disabled=true)
  p2003sub0 (Disabled=true)
  p2003sub0_parametername =  (Disabled=true)
  p2003sub0_objecttype =  (Disabled=true)
  p2003sub0_datatype =  (Disabled=true)
  p2003sub0_accesstype =  (Disabled=true)
  p2003sub0_pdomapping =  (Disabled=true)
  p2003sub0_parametervalue =  (Disabled=true)
  p2003sub0_objflags = 1 (Disabled=true)
  p2003sub1 (Disabled=true)
  p2003sub1_parametername =  (Disabled=true)
  p2003sub1_objecttype =  (Disabled=true)
  p2003sub1_datatype =  (Disabled=true)
  p2003sub1_accesstype =  (Disabled=true)
  p2003sub1_pdomapping =  (Disabled=true)
  p2003sub1_highlimit =  (Disabled=true)
  p2003sub1_parametervalue =  (Disabled=true)
  p2003sub1_objflags = 1 (Disabled=true)
  p2003sub2 (Disabled=true)
  p2003sub2_parametername =  (Disabled=true)
  p2003sub2_objecttype =  (Disabled=true)
  p2003sub2_datatype =  (Disabled=true)
  p2003sub2_accesstype =  (Disabled=true)
  p2003sub2_pdomapping =  (Disabled=true)
  p2003sub2_parametervalue =  (Disabled=true)
  p2003sub2_objflags = 1 (Disabled=true)
  p2003sub3 (Disabled=true)
  p2003sub3_parametername =  (Disabled=true)
  p2003sub3_objecttype =  (Disabled=true)
  p2003sub3_datatype =  (Disabled=true)
  p2003sub3_accesstype =  (Disabled=true)
  p2003sub3_pdomapping =  (Disabled=true)
  p2003sub3_highlimit =  (Disabled=true)
  p2003sub3_parametervalue =  (Disabled=true)
  p2003sub3_objflags = 1 (Disabled=true)
  p2004 (Disabled=true)
  p2004_parametername =  (Disabled=true)
  p2004_objecttype =  (Disabled=true)
  p2004_datatype =  (Disabled=true)
  p2004_accesstype =  (Disabled=true)
  p2004_pdomapping =  (Disabled=true)
  p2004_parametervalue =  (Disabled=true)
  p2004_objflags = 1 (Disabled=true)
  p2005 (Disabled=true)
  p2005_parametername =  (Disabled=true)
  p2005_objecttype =  (Disabled=true)
  p2005_datatype =  (Disabled=true)
  p2005_subnumber =  (Disabled=true)
  p2005_parametervalue =  (Disabled=true)
  p2005_objflags = 1 (Disabled=true)
  p2005sub0 (Disabled=true)
  p2005sub0_parametername =  (Disabled=true)
  p2005sub0_objecttype =  (Disabled=true)
  p2005sub0_datatype =  (Disabled=true)
  p2005sub0_accesstype =  (Disabled=true)
  p2005sub0_pdomapping =  (Disabled=true)
  p2005sub0_parametervalue =  (Disabled=true)
  p2005sub0_objflags = 1 (Disabled=true)
  p2005sub1 (Disabled=true)
  p2005sub1_parametername =  (Disabled=true)
  p2005sub1_objecttype =  (Disabled=true)
  p2005sub1_datatype =  (Disabled=true)
  p2005sub1_accesstype =  (Disabled=true)
  p2005sub1_pdomapping =  (Disabled=true)
  p2005sub1_highlimit =  (Disabled=true)
  p2005sub1_parametervalue =  (Disabled=true)
  p2005sub1_objflags = 1 (Disabled=true)
  p2005sub2 (Disabled=true)
  p2005sub2_parametername =  (Disabled=true)
  p2005sub2_objecttype =  (Disabled=true)
  p2005sub2_datatype =  (Disabled=true)
  p2005sub2_accesstype =  (Disabled=true)
  p2005sub2_pdomapping =  (Disabled=true)
  p2005sub2_highlimit =  (Disabled=true)
  p2005sub2_parametervalue =  (Disabled=true)
  p2005sub2_objflags = 1 (Disabled=true)
  p2005sub3 (Disabled=true)
  p2005sub3_parametername =  (Disabled=true)
  p2005sub3_objecttype =  (Disabled=true)
  p2005sub3_datatype =  (Disabled=true)
  p2005sub3_accesstype =  (Disabled=true)
  p2005sub3_pdomapping =  (Disabled=true)
  p2005sub3_highlimit =  (Disabled=true)
  p2005sub3_parametervalue =  (Disabled=true)
  p2005sub3_objflags = 1 (Disabled=true)
  p2005sub4 (Disabled=true)
  p2005sub4_parametername =  (Disabled=true)
  p2005sub4_objecttype =  (Disabled=true)
  p2005sub4_datatype =  (Disabled=true)
  p2005sub4_accesstype =  (Disabled=true)
  p2005sub4_pdomapping =  (Disabled=true)
  p2005sub4_highlimit =  (Disabled=true)
  p2005sub4_parametervalue =  (Disabled=true)
  p2005sub4_objflags = 1 (Disabled=true)
  p2006 (Disabled=true)
  p2006_parametername =  (Disabled=true)
  p2006_objecttype =  (Disabled=true)
  p2006_datatype =  (Disabled=true)
  p2006_accesstype =  (Disabled=true)
  p2006_pdomapping =  (Disabled=true)
  p2006_highlimit =  (Disabled=true)
  p2006_parametervalue = 1112276992 (Disabled=true)
  p2006_objflags = 1 (Disabled=true)
  p2007 (Disabled=true)
  p2007_parametername =  (Disabled=true)
  p2007_objecttype =  (Disabled=true)
  p2007_datatype =  (Disabled=true)
  p2007_accesstype =  (Disabled=true)
  p2007_pdomapping =  (Disabled=true)
  p2007_highlimit =  (Disabled=true)
  p2007_parametervalue =  (Disabled=true)
  p2007_objflags = 1 (Disabled=true)
  p2008 (Disabled=true)
  p2008_parametername =  (Disabled=true)
  p2008_objecttype =  (Disabled=true)
  p2008_datatype =  (Disabled=true)
  p2008_accesstype =  (Disabled=true)
  p2008_pdomapping =  (Disabled=true)
  p2008_highlimit =  (Disabled=true)
  p2008_parametervalue =  (Disabled=true)
  p2008_objflags = 1 (Disabled=true)
  p2009 (Disabled=true)
  p2009_parametername =  (Disabled=true)
  p2009_objecttype =  (Disabled=true)
  p2009_datatype =  (Disabled=true)
  p2009_subnumber =  (Disabled=true)
  p2009_parametervalue =  (Disabled=true)
  p2009_objflags = 1 (Disabled=true)
  p2009sub0 (Disabled=true)
  p2009sub0_parametername =  (Disabled=true)
  p2009sub0_objecttype =  (Disabled=true)
  p2009sub0_datatype =  (Disabled=true)
  p2009sub0_accesstype =  (Disabled=true)
  p2009sub0_pdomapping =  (Disabled=true)
  p2009sub0_parametervalue =  (Disabled=true)
  p2009sub0_objflags = 1 (Disabled=true)
  p2009sub1 (Disabled=true)
  p2009sub1_parametername =  (Disabled=true)
  p2009sub1_objecttype =  (Disabled=true)
  p2009sub1_datatype =  (Disabled=true)
  p2009sub1_accesstype =  (Disabled=true)
  p2009sub1_pdomapping =  (Disabled=true)
  p2009sub1_highlimit =  (Disabled=true)
  p2009sub1_parametervalue = 0 (Disabled=true)
  p2009sub1_objflags = 1 (Disabled=true)
  p2009sub2 (Disabled=true)
  p2009sub2_parametername =  (Disabled=true)
  p2009sub2_objecttype =  (Disabled=true)
  p2009sub2_datatype =  (Disabled=true)
  p2009sub2_accesstype =  (Disabled=true)
  p2009sub2_pdomapping =  (Disabled=true)
  p2009sub2_highlimit =  (Disabled=true)
  p2009sub2_parametervalue = 0 (Disabled=true)
  p2009sub2_objflags = 1 (Disabled=true)
  p200a (Disabled=true)
  p200a_parametername =  (Disabled=true)
  p200a_objecttype =  (Disabled=true)
  p200a_datatype =  (Disabled=true)
  p200a_subnumber =  (Disabled=true)
  p200a_parametervalue =  (Disabled=true)
  p200a_objflags = 1 (Disabled=true)
  p200asub0 (Disabled=true)
  p200asub0_parametername =  (Disabled=true)
  p200asub0_objecttype =  (Disabled=true)
  p200asub0_datatype =  (Disabled=true)
  p200asub0_accesstype =  (Disabled=true)
  p200asub0_pdomapping =  (Disabled=true)
  p200asub0_parametervalue =  (Disabled=true)
  p200asub0_objflags = 1 (Disabled=true)
  p200asub1 (Disabled=true)
  p200asub1_parametername =  (Disabled=true)
  p200asub1_objecttype =  (Disabled=true)
  p200asub1_datatype =  (Disabled=true)
  p200asub1_accesstype =  (Disabled=true)
  p200asub1_pdomapping =  (Disabled=true)
  p200asub1_highlimit =  (Disabled=true)
  p200asub1_parametervalue = 1092616192 (Disabled=true)
  p200asub1_objflags = 1 (Disabled=true)
  p200asub2 (Disabled=true)
  p200asub2_parametername =  (Disabled=true)
  p200asub2_objecttype =  (Disabled=true)
  p200asub2_datatype =  (Disabled=true)
  p200asub2_accesstype =  (Disabled=true)
  p200asub2_pdomapping =  (Disabled=true)
  p200asub2_highlimit =  (Disabled=true)
  p200asub2_parametervalue = 1092616192 (Disabled=true)
  p200asub2_objflags = 1 (Disabled=true)
  p200b (Disabled=true)
  p200b_parametername =  (Disabled=true)
  p200b_objecttype =  (Disabled=true)
  p200b_datatype =  (Disabled=true)
  p200b_subnumber =  (Disabled=true)
  p200b_parametervalue =  (Disabled=true)
  p200b_objflags = 1 (Disabled=true)
  p200bsub0 (Disabled=true)
  p200bsub0_parametername =  (Disabled=true)
  p200bsub0_objecttype =  (Disabled=true)
  p200bsub0_datatype =  (Disabled=true)
  p200bsub0_accesstype =  (Disabled=true)
  p200bsub0_pdomapping =  (Disabled=true)
  p200bsub0_parametervalue =  (Disabled=true)
  p200bsub0_objflags = 1 (Disabled=true)
  p200bsub1 (Disabled=true)
  p200bsub1_parametername =  (Disabled=true)
  p200bsub1_objecttype =  (Disabled=true)
  p200bsub1_datatype =  (Disabled=true)
  p200bsub1_accesstype =  (Disabled=true)
  p200bsub1_pdomapping =  (Disabled=true)
  p200bsub1_highlimit =  (Disabled=true)
  p200bsub1_parametervalue = 1036831949 (Disabled=true)
  p200bsub1_objflags = 1 (Disabled=true)
  p200bsub2 (Disabled=true)
  p200bsub2_parametername =  (Disabled=true)
  p200bsub2_objecttype =  (Disabled=true)
  p200bsub2_datatype =  (Disabled=true)
  p200bsub2_accesstype =  (Disabled=true)
  p200bsub2_pdomapping =  (Disabled=true)
  p200bsub2_highlimit =  (Disabled=true)
  p200bsub2_parametervalue = 0 (Disabled=true)
  p200bsub2_objflags = 1 (Disabled=true)
  p200c (Disabled=true)
  p200c_parametername =  (Disabled=true)
  p200c_objecttype =  (Disabled=true)
  p200c_datatype =  (Disabled=true)
  p200c_subnumber =  (Disabled=true)
  p200c_parametervalue =  (Disabled=true)
  p200c_objflags = 1 (Disabled=true)
  p200csub0 (Disabled=true)
  p200csub0_parametername =  (Disabled=true)
  p200csub0_objecttype =  (Disabled=true)
  p200csub0_datatype =  (Disabled=true)
  p200csub0_accesstype =  (Disabled=true)
  p200csub0_pdomapping =  (Disabled=true)
  p200csub0_parametervalue =  (Disabled=true)
  p200csub0_objflags = 1 (Disabled=true)
  p200csub1 (Disabled=true)
  p200csub1_parametername =  (Disabled=true)
  p200csub1_objecttype =  (Disabled=true)
  p200csub1_datatype =  (Disabled=true)
  p200csub1_accesstype =  (Disabled=true)
  p200csub1_pdomapping =  (Disabled=true)
  p200csub1_highlimit =  (Disabled=true)
  p200csub1_parametervalue = 1008981770 (Disabled=true)
  p200csub1_objflags = 1 (Disabled=true)
  p200csub2 (Disabled=true)
  p200csub2_parametername =  (Disabled=true)
  p200csub2_objecttype =  (Disabled=true)
  p200csub2_datatype =  (Disabled=true)
  p200csub2_accesstype =  (Disabled=true)
  p200csub2_pdomapping =  (Disabled=true)
  p200csub2_highlimit =  (Disabled=true)
  p200csub2_parametervalue = 0 (Disabled=true)
  p200csub2_objflags = 1 (Disabled=true)
  p200d (Disabled=true)
  p200d_parametername =  (Disabled=true)
  p200d_objecttype =  (Disabled=true)
  p200d_datatype =  (Disabled=true)
  p200d_subnumber =  (Disabled=true)
  p200d_parametervalue =  (Disabled=true)
  p200d_objflags = 1 (Disabled=true)
  p200dsub0 (Disabled=true)
  p200dsub0_parametername =  (Disabled=true)
  p200dsub0_objecttype =  (Disabled=true)
  p200dsub0_datatype =  (Disabled=true)
  p200dsub0_accesstype =  (Disabled=true)
  p200dsub0_pdomapping =  (Disabled=true)
  p200dsub0_parametervalue =  (Disabled=true)
  p200dsub0_objflags = 1 (Disabled=true)
  p200dsub1 (Disabled=true)
  p200dsub1_parametername =  (Disabled=true)
  p200dsub1_objecttype =  (Disabled=true)
  p200dsub1_datatype =  (Disabled=true)
  p200dsub1_accesstype =  (Disabled=true)
  p200dsub1_pdomapping =  (Disabled=true)
  p200dsub1_highlimit =  (Disabled=true)
  p200dsub1_parametervalue =  (Disabled=true)
  p200dsub1_objflags = 1 (Disabled=true)
  p200dsub2 (Disabled=true)
  p200dsub2_parametername =  (Disabled=true)
  p200dsub2_objecttype =  (Disabled=true)
  p200dsub2_datatype =  (Disabled=true)
  p200dsub2_accesstype =  (Disabled=true)
  p200dsub2_pdomapping =  (Disabled=true)
  p200dsub2_highlimit =  (Disabled=true)
  p200dsub2_parametervalue =  (Disabled=true)
  p200dsub2_objflags = 1 (Disabled=true)
  p200e (Disabled=true)
  p200e_parametername =  (Disabled=true)
  p200e_objecttype =  (Disabled=true)
  p200e_datatype =  (Disabled=true)
  p200e_subnumber =  (Disabled=true)
  p200e_parametervalue =  (Disabled=true)
  p200e_objflags = 1 (Disabled=true)
  p200esub0 (Disabled=true)
  p200esub0_parametername =  (Disabled=true)
  p200esub0_objecttype =  (Disabled=true)
  p200esub0_datatype =  (Disabled=true)
  p200esub0_accesstype =  (Disabled=true)
  p200esub0_pdomapping =  (Disabled=true)
  p200esub0_parametervalue =  (Disabled=true)
  p200esub0_objflags = 1 (Disabled=true)
  p200f (Disabled=true)
  p200f_parametername =  (Disabled=true)
  p200f_objecttype =  (Disabled=true)
  p200f_datatype =  (Disabled=true)
  p200f_accesstype =  (Disabled=true)
  p200f_pdomapping =  (Disabled=true)
  p200f_highlimit =  (Disabled=true)
  p200f_parametervalue =  (Disabled=true)
  p200f_objflags = 1 (Disabled=true)
  p2010 (Disabled=true)
  p2010_parametername =  (Disabled=true)
  p2010_objecttype =  (Disabled=true)
  p2010_datatype =  (Disabled=true)
  p2010_accesstype =  (Disabled=true)
  p2010_pdomapping =  (Disabled=true)
  p2010_highlimit =  (Disabled=true)
  p2010_parametervalue =  (Disabled=true)
  p2010_objflags = 1 (Disabled=true)
  p2011 (Disabled=true)
  p2011_parametername =  (Disabled=true)
  p2011_objecttype =  (Disabled=true)
  p2011_datatype =  (Disabled=true)
  p2011_accesstype =  (Disabled=true)
  p2011_pdomapping =  (Disabled=true)
  p2011_highlimit =  (Disabled=true)
  p2011_parametervalue =  (Disabled=true)
  p2011_objflags = 1 (Disabled=true)
  p2012 (Disabled=true)
  p2012_parametername =  (Disabled=true)
  p2012_objecttype =  (Disabled=true)
  p2012_datatype =  (Disabled=true)
  p2012_subnumber =  (Disabled=true)
  p2012_parametervalue =  (Disabled=true)
  p2012_objflags = 1 (Disabled=true)
  p2012sub0 (Disabled=true)
  p2012sub0_parametername =  (Disabled=true)
  p2012sub0_objecttype =  (Disabled=true)
  p2012sub0_datatype =  (Disabled=true)
  p2012sub0_accesstype =  (Disabled=true)
  p2012sub0_parametervalue =  (Disabled=true)
  p2012sub0_objflags = 1 (Disabled=true)
  p2012sub1 (Disabled=true)
  p2012sub1_parametername =  (Disabled=true)
  p2012sub1_objecttype =  (Disabled=true)
  p2012sub1_datatype =  (Disabled=true)
  p2012sub1_accesstype =  (Disabled=true)
  p2012sub1_pdomapping =  (Disabled=true)
  p2012sub1_highlimit =  (Disabled=true)
  p2012sub1_parametervalue = 0 (Disabled=true)
  p2012sub1_objflags = 1 (Disabled=true)
  p2012sub2 (Disabled=true)
  p2012sub2_parametername =  (Disabled=true)
  p2012sub2_objecttype =  (Disabled=true)
  p2012sub2_datatype =  (Disabled=true)
  p2012sub2_accesstype =  (Disabled=true)
  p2012sub2_pdomapping =  (Disabled=true)
  p2012sub2_highlimit =  (Disabled=true)
  p2012sub2_parametervalue = 0 (Disabled=true)
  p2012sub2_objflags = 1 (Disabled=true)
  p2012sub3 (Disabled=true)
  p2012sub3_parametername =  (Disabled=true)
  p2012sub3_objecttype =  (Disabled=true)
  p2012sub3_datatype =  (Disabled=true)
  p2012sub3_accesstype =  (Disabled=true)
  p2012sub3_pdomapping =  (Disabled=true)
  p2012sub3_highlimit =  (Disabled=true)
  p2012sub3_parametervalue = 0 (Disabled=true)
  p2012sub3_objflags = 1 (Disabled=true)
  p2012sub4 (Disabled=true)
  p2012sub4_parametername =  (Disabled=true)
  p2012sub4_objecttype =  (Disabled=true)
  p2012sub4_datatype =  (Disabled=true)
  p2012sub4_accesstype =  (Disabled=true)
  p2012sub4_pdomapping =  (Disabled=true)
  p2012sub4_highlimit =  (Disabled=true)
  p2012sub4_parametervalue = 0 (Disabled=true)
  p2012sub4_objflags = 1 (Disabled=true)
  p2012sub5 (Disabled=true)
  p2012sub5_parametername =  (Disabled=true)
  p2012sub5_objecttype =  (Disabled=true)
  p2012sub5_datatype =  (Disabled=true)
  p2012sub5_accesstype =  (Disabled=true)
  p2012sub5_pdomapping =  (Disabled=true)
  p2012sub5_highlimit =  (Disabled=true)
  p2012sub5_parametervalue = 0 (Disabled=true)
  p2012sub5_objflags = 1 (Disabled=true)
  p6075 (Disabled=true)
  p6075_parametername =  (Disabled=true)
  p6075_objecttype =  (Disabled=true)
  p6075_datatype =  (Disabled=true)
  p6075_accesstype =  (Disabled=true)
  p6075_pdomapping =  (Disabled=true)
  p6075_parametervalue =  (Disabled=true)
  p6075_objflags = 1 (Disabled=true)
  p607b (Disabled=true)
  p607b_parametername =  (Disabled=true)
  p607b_objecttype =  (Disabled=true)
  p607b_datatype =  (Disabled=true)
  p607b_subnumber =  (Disabled=true)
  p607b_parametervalue =  (Disabled=true)
  p607b_objflags = 1 (Disabled=true)
  p607bsub0 (Disabled=true)
  p607bsub0_parametername =  (Disabled=true)
  p607bsub0_objecttype =  (Disabled=true)
  p607bsub0_datatype =  (Disabled=true)
  p607bsub0_accesstype =  (Disabled=true)
  p607bsub0_pdomapping =  (Disabled=true)
  p607bsub0_parametervalue =  (Disabled=true)
  p607bsub0_objflags = 1 (Disabled=true)
  p608f (Disabled=true)
  p608f_parametername =  (Disabled=true)
  p608f_objecttype =  (Disabled=true)
  p608f_subnumber =  (Disabled=true)
  p608f_parametervalue =  (Disabled=true)
  p608f_objflags = 1 (Disabled=true)
  p608fsub0 (Disabled=true)
  p608fsub0_parametername =  (Disabled=true)
  p608fsub0_objecttype =  (Disabled=true)
  p608fsub0_datatype =  (Disabled=true)
  p608fsub0_accesstype =  (Disabled=true)
  p608fsub0_pdomapping =  (Disabled=true)
  p608fsub0_parametervalue =  (Disabled=true)
  p608fsub0_objflags = 1 (Disabled=true)
  p6091 (Disabled=true)
  p6091_parametername =  (Disabled=true)
  p6091_objecttype =  (Disabled=true)
  p6091_subnumber =  (Disabled=true)
  p6091_parametervalue =  (Disabled=true)
  p6091_objflags = 1 (Disabled=true)
  p6091sub0 (Disabled=true)
  p6091sub0_parametername =  (Disabled=true)
  p6091sub0_objecttype =  (Disabled=true)
  p6091sub0_datatype =  (Disabled=true)
  p6091sub0_accesstype =  (Disabled=true)
  p6091sub0_pdomapping =  (Disabled=true)
  p6091sub0_parametervalue =  (Disabled=true)
  p6091sub0_objflags = 1 (Disabled=true)
  p6092 (Disabled=true)
  p6092_parametername =  (Disabled=true)
  p6092_objecttype =  (Disabled=true)
  p6092_subnumber =  (Disabled=true)
  p6092_parametervalue =  (Disabled=true)
  p6092_objflags = 1 (Disabled=true)
  p6092sub0 (Disabled=true)
  p6092sub0_parametername =  (Disabled=true)
  p6092sub0_objecttype =  (Disabled=true)
  p6092sub0_datatype =  (Disabled=true)
  p6092sub0_accesstype =  (Disabled=true)
  p6092sub0_pdomapping =  (Disabled=true)
  p6092sub0_parametervalue =  (Disabled=true)
  p6092sub0_objflags = 1 (Disabled=true)
  p6099 (Disabled=true)
  p6099_parametername =  (Disabled=true)
  p6099_objecttype =  (Disabled=true)
  p6099_subnumber =  (Disabled=true)
  p6099_parametervalue =  (Disabled=true)
  p6099_objflags = 1 (Disabled=true)
  p6099sub0 (Disabled=true)
  p6099sub0_parametername =  (Disabled=true)
  p6099sub0_objecttype =  (Disabled=true)
  p6099sub0_datatype =  (Disabled=true)
  p6099sub0_accesstype =  (Disabled=true)
  p6099sub0_pdomapping =  (Disabled=true)
  p6099sub0_parametervalue =  (Disabled=true)
  p6099sub0_objflags = 1 (Disabled=true)
  p60a8 (Disabled=true)
  p60a8_parametername =  (Disabled=true)
  p60a8_objecttype =  (Disabled=true)
  p60a8_datatype =  (Disabled=true)
  p60a8_accesstype =  (Disabled=true)
  p60a8_pdomapping =  (Disabled=true)
  p60a8_parametervalue =  (Disabled=true)
  p60a8_objflags = 1 (Disabled=true)
  p60c2 (Disabled=true)
  p60c2_parametername =  (Disabled=true)
  p60c2_objecttype =  (Disabled=true)
  p60c2_subnumber =  (Disabled=true)
  p60c2_parametervalue =  (Disabled=true)
  p60c2_objflags = 1 (Disabled=true)
  p60c2sub0 (Disabled=true)
  p60c2sub0_parametername =  (Disabled=true)
  p60c2sub0_objecttype =  (Disabled=true)
  p60c2sub0_datatype =  (Disabled=true)
  p60c2sub0_accesstype =  (Disabled=true)
  p60c2sub0_pdomapping =  (Disabled=true)
  p60c2sub0_parametervalue =  (Disabled=true)
  p60c2sub0_objflags = 1 (Disabled=true)
  p60fe (Disabled=true)
  p60fe_parametername =  (Disabled=true)
  p60fe_objecttype =  (Disabled=true)
  p60fe_subnumber =  (Disabled=true)
  p60fe_parametervalue =  (Disabled=true)
  p60fe_objflags = 1 (Disabled=true)
  p60fesub0 (Disabled=true)
  p60fesub0_parametername =  (Disabled=true)
  p60fesub0_objecttype =  (Disabled=true)
  p60fesub0_datatype =  (Disabled=true)
  p60fesub0_accesstype =  (Disabled=true)
  p60fesub0_pdomapping =  (Disabled=true)
  p60fesub0_parametervalue =  (Disabled=true)
  p60fesub0_objflags = 1 (Disabled=true)
  p6402 (Disabled=true)
  p6402_parametername =  (Disabled=true)
  p6402_objecttype =  (Disabled=true)
  p6402_datatype =  (Disabled=true)
  p6402_accesstype =  (Disabled=true)
  p6402_pdomapping =  (Disabled=true)
  p6402_parametervalue =  (Disabled=true)
  p6402_objflags = 1 (Disabled=true)
```

### IoMap.iom - 5PPC2100_BY34_000/IoMap.iom
```iecst
VAR_CONFIG
	glb_drv.out.ContolWord6040 AT %QW."dryve-D1".Controlword_6040;
	glb_drv.inp.StatusWord6041 AT %IW."dryve-D1".Statusword_6041;
	glb_drv.inp.PositionActualValue6064 AT %ID."dryve-D1".PositionActualValue_6064;
	glb_drv.inp.VelocityActualValue606C AT %ID."dryve-D1".VelocityActualValue_606C;
	glb_drv.out.TargetPosition607A AT %QD."dryve-D1".TargetPosition_607A;
	glb_drv.out.TargetVelocity60FF AT %QD."dryve-D1".TargetVelocity_60FF;
	glb_drv.inp.ErrorCode_603f AT %IW."dryve-D1".ErrorCode_603F;
	glb_drv.out.ModesOfOperation_6060 AT %QB."dryve-D1".ModesOfOperation_6060;
	glb_drv.inp.ModesOfOperationDisplay_6061 AT %IB."dryve-D1".ModesOfOperationDisplay_6061;
	glb_drv.out.ProfileVelocity6081 AT %QD."dryve-D1".ProfileVelocity_6081;
	glb_drv.out.ProfileAcceleration6083 AT %QD."dryve-D1".ProfileAcceleration_6083;
	glb_drv.out.HomingAcceleration609A AT %QD."dryve-D1".HomingAcceleration_609A;
	glb_drv.out.HomeHighSpeed6099_sub1 AT %QD."dryve-D1".HomingSpeedsSpeedDuringSearchForSwitch_6099sub1;
	glb_drv.out.HomeLowSpeed6099_sub2 AT %QD."dryve-D1".HomingSpeedsSpeedDuringSearchForZero_6099sub2;
	glb_drv.out.FeedConstantFeed6092_sub1 AT %QD."dryve-D1".FeedConstantFeed_6092sub1;
	glb_drv.out.FeedConstantShaftRev6092_sub2 AT %QD."dryve-D1".FeedConstantShaftRevolutions_6092sub2;
END_VAR
```

### Config.mprecipexml - 5PPC2100_BY34_000/mappServices/Config.mprecipexml
```
Element gRecipeXml (Type=mprecipexml)
```

## Logical view

Binary libraries used (declarations not repeated): operator, runtime, astime, AsIecCon, McBase, MpAxis 5.12.2, AsTCP, standard, asstring, sys_lib, FileIO, MpAlarmX 5.24.1, MpBase, MpFile 5.24.1, MpRecipe 5.24.1, Acp10par 5.24.1, AsIOAcc, AsIORTI, AsMath, MpUser 5.24.1, NcGlobal 5.24.1

### Global.typ - Global data types
```iecst
TYPE
	typ_tcp_state : 	STRUCT
		tcpopen : BOOL;
		tcpioctl : BOOL;
		tcpclient : BOOL;
		tcpsend : BOOL;
		tcprecv : BOOL;
		tcpclose : BOOL;
		tcperror : BOOL;
	END_STRUCT;
	typ_tcp_protocol_state : 	STRUCT
		place_older : BOOL;
	END_STRUCT;
	typ_io : 	STRUCT
		Do : typ_Do;
		Di : typ_Di;
	END_STRUCT;
	typ_eth_connect : 	STRUCT
		machine_in_auto : BOOL;
		machine_in_man : BOOL;
		machine_stopped : BOOL;
		machine_in_error : BOOL;
		stop_request : BOOL; (*Richiesta di stop*)
		last_cycle_request : BOOL; (*Richiesta di fermarsi dopo il ciclo attuale*)
		step : USINT;
		counter : UINT; (*Contatore*)
		no_comunication : BOOL; (*No comunication with master device*)
		protocol_state : typ_tcp_protocol_state; (*Stato della sincronizzazione*)
		tcp_state : typ_tcp_state; (*Stato della comunicazione tcp*)
		disable : BOOL; (*Disabilito il protocollo di comunicazione*)
		Server_Ip_Add : STRING[15] := '192.168.250.15';
	END_STRUCT;
	typ_drv_out : 	STRUCT
		ContolWord6040 : UINT;
		ModesOfOperation_6060 : SINT;
		TargetTorque_6071 : INT;
		TargetPosition607A : DINT;
		FollowingErrorWindow6065 : DINT;
		PositionWindow6067 : DINT;
		PositionWindowTime6068 : INT;
		ProfileVelocity6081 : UDINT;
		ProfileAcceleration6083 : UDINT;
		ProfileDeceleration6084 : UDINT;
		PositonFactor6093_sub1 : UDINT;
		PositonFactor6093_sub2 : UDINT;
		TorqueSlope_6087 : UDINT;
		HomingMethod6098 : SINT;
		HomeOffset607C : DINT;
		HomeHighSpeed6099_sub1 : UDINT;
		HomeLowSpeed6099_sub2 : UDINT;
		HomingAcceleration609A : UDINT;
		TargetVelocity60FF : DINT;
		FeedConstantFeed6092_sub1 : UDINT;
		FeedConstantShaftRev6092_sub2 : UDINT;
		DRV_ON_CMD : BOOL; (*BIT 0 DELLA CONTROL WORD 6040*)
		DRV_ENABLE_VOLT_CMD : BOOL; (*BIT 1 DELLA CONTROL WORD 6040*)
		DRV_QUICK_STOP_CMD : BOOL; (*BIT 2 DELLA CONTROL WORD 6040*)
		DRV_EN_OP_CMD : BOOL; (*BIT 3 DELLA CONTROL WORD 6040*)
		DRV_START_HM_NEW_PP_CMD : BOOL; (*BIT 4 DELLA CONTROL WORD 6040 (NOTA BENE: IN HM VALE HOMING OPERATION START POSITIVE TRIGGER; IN PROFILE POSITION MODE VALE "NEW SETPOINT [POSITIVE TRIGGER]"*)
		DRV_CHANGE_SET_IMM : BOOL; (*BIT 5 DELLA CONTROL WORD 6040-FUNZIONA SOLO CON IL PROFILE POSITION E SERVE PER SETTARE IMMEDIATAMENTE LA POSIZIONE*)
		DRV_TOGGLE_ABS_REL : BOOL; (*BIT 6 DELLA CONTROL WORD 6040- 0=ASSOLUTO; 1=RELATIVO (ENCODER?)*)
		DRV_FAULT_RESET_CMD : BOOL; (*BIT 7 DELLA CONTROL WORD 6040*)
		DRV_HALT_CMD : BOOL; (*BIT 8 DELLA CONTROL WORD 6040*)
	END_STRUCT;
	typ_drv_inp : 	STRUCT
		DRV_READY : BOOL;
		DRV_ON : BOOL;
		DRV_OPERATION_ENABLED : BOOL;
		DRV_FAULT : BOOL;
		DRV_VOLT_ENABLE : BOOL;
		DRV_SWITCH_ON_DISABLED : BOOL;
		DRV_WARNING : BOOL;
		DRV_REMOTE : BOOL;
		DRV_TARGET_REACHED : BOOL;
		DRV_TARGET_STATUS : BOOL;
		DRV_MOVE_ERROR : BOOL;
		DRV_QUICK_STOP : BOOL;
		StatusWord6041 : UINT;
		ModesOfOperationDisplay_6061 : SINT;
		PositionActualValue6064 : DINT;
		VelocityActualValue606C : DINT;
		TorqueDemandValue_6074 : INT;
		MotorRatedCurrent_6075 : UDINT;
		TorqueActualValue_6077 : INT;
		CurrentActualValue_6078 : INT;
		ErrorCode_603f : UINT;
	END_STRUCT;
	typ_drv : 	STRUCT
		inp : typ_drv_inp;
		out : typ_drv_out;
	END_STRUCT;
	typ_Do : 	STRUCT
		Piston_up : BOOL;
		Piston_gun_2 : BOOL;
		Piston_gun_1 : BOOL;
	END_STRUCT;
	typ_Di : 	STRUCT
		Finecorsa : BOOL;
		Si_01 : BOOL;
		Si_02 : BOOL;
		Start : BOOL;
		Stop : BOOL;
		Automatic : BOOL;
	END_STRUCT;
	En_status :
		(
		STOP := 0,
		AUTO := 10,
		MANUAL := 20,
		ERR := 30
		);
END_TYPE
```

### Global.var - Global variables
```iecst
VAR
	Ricetta : USINT;
	Status : En_status;
	glb_io : typ_io;
	glb_drv : typ_drv;
	Eth_connect : typ_eth_connect;
END_VAR
```

### Constant.var
```iecst
VAR CONSTANT
	bit_0 : UINT := 1;
	bit_1 : UINT := 2;
	bit_2 : UINT := 4;
	bit_3 : UINT := 8;
	bit_4 : UINT := 16;
	bit_5 : UINT := 32;
	bit_6 : UINT := 64;
	bit_7 : UINT := 128;
	bit_8 : UINT := 256;
	bit_9 : UDINT := 512;
	bit_10 : UDINT := 1024;
	bit_11 : UDINT := 2048;
	bit_12 : UDINT := 4096;
	bit_13 : UDINT := 8192;
	bit_14 : UDINT := 16384;
	bit_15 : UDINT := 32768;
	bit_16 : UDINT := 65536;
	bit_17 : UDINT := 131072;
	bit_18 : UDINT := 262144;
	bit_19 : UDINT := 524288;
	bit_20 : UDINT := 1048576;
	bit_21 : UDINT := 2097152;
	bit_22 : UDINT := 4194304;
	bit_23 : UDINT := 8388608;
	bit_24 : UDINT := 16777216;
	bit_25 : UDINT := 33554432;
	bit_26 : UDINT := 67108864;
	bit_27 : UDINT := 134217728;
	bit_28 : UDINT := 268435456;
	bit_29 : UDINT := 536870912;
	bit_30 : UDINT := 1073741824;
	bit_31 : UDINT := 2147483648;
	bit_negato_0 : UDINT := 4294967294;
	bit_negato_1 : UDINT := 4294967293;
	bit_negato_2 : UDINT := 4294967291;
	bit_negato_3 : UDINT := 4294967287;
	bit_negato_4 : UDINT := 4294967279;
	bit_negato_5 : UDINT := 4294967263;
	bit_negato_6 : UDINT := 4294967231;
	bit_negato_7 : UDINT := 4294967167;
	bit_negato_8 : UDINT := 4294967039;
	bit_negato_9 : UDINT := 4294966783;
	bit_negato_10 : UDINT := 4294966271;
	bit_negato_11 : UDINT := 4294965247;
	bit_negato_12 : UDINT := 4294963199;
	bit_negato_13 : UDINT := 4294959103;
	bit_negato_14 : UDINT := 4294950911;
	bit_negato_15 : UDINT := 4294934527;
	bit_negato_16 : UDINT := 4294901759;
	bit_negato_17 : UDINT := 4294836223;
	bit_negato_18 : UDINT := 4294705151;
	bit_negato_19 : UDINT := 4294443007;
	bit_negato_20 : UDINT := 4293918719;
	bit_negato_21 : UDINT := 4292870143;
	bit_negato_22 : UDINT := 4290772991;
	bit_negato_23 : UDINT := 4286578687;
	bit_negato_24 : UDINT := 4278190079;
	bit_negato_25 : UDINT := 4261412863;
	bit_negato_26 : UDINT := 4227858431;
	bit_negato_27 : UDINT := 4160749567;
	bit_negato_28 : UDINT := 4026531839;
	bit_negato_29 : UDINT := 3758096383;
	bit_negato_30 : UDINT := 3221225471;
	bit_negato_31 : UDINT := 2147483647;
	UINT_negato_0 : UINT := 65534;
	UINT_negato_1 : UINT := 65533;
	UINT_negato_2 : UINT := 65531;
	UINT_negato_3 : UINT := 65527;
	UINT_negato_4 : UINT := 65519;
	UINT_negato_5 : UINT := 65503;
	UINT_negato_6 : UINT := 65471;
	UINT_negato_7 : UINT := 65407;
	UINT_negato_8 : UINT := 65279;
END_VAR
```

### Package Logical/Libraries - Global libraries

### Library Logical/Libraries/XSM_Ramp (IEC, version 1.00.5)
Depends on: brsystem, AsIOAcc, asstring, AsMath

#### XSM_Ramp.fun
```iecst
FUNCTION_BLOCK XSM_Ctrl (*Stepper motor control*)
	VAR_INPUT
		Enable : BOOL;
		Power : BOOL;
		Cmd : XSM_Ctrl_CmdType;
		IO_Mapping : XSM_Ctrl_IOMappingType;
		Parameters : XSM_Ctrl_ParametersType;
	END_VAR
	VAR_OUTPUT
		Active : BOOL;
		PowerOn : BOOL;
		Error : BOOL;
		Status : UINT;
		Monitor : XSM_Ctrl_MonitorType;
	END_VAR
	VAR
		intern : XSM_Ctrl_internType;
		RTInfo_0 : RTInfo;
		AsIOAccRead_0 : AsIOAccRead;
		AsIOAccReadReg_0 : AsIOAccReadReg;
		zzEdge00000 : BOOL;
	END_VAR
END_FUNCTION_BLOCK

FUNCTION_BLOCK XSM_IO_Cfg (*Configure stepper motor IO configuration.*)
	VAR_INPUT
		Enable : BOOL;
		Config : BOOL;
		Mode : USINT;
		Reset : BOOL;
		IO_Cfg : XSM_IO_ConfigurationType;
		pIO_Mapping : UDINT;
		pParameters : UDINT;
	END_VAR
	VAR_OUTPUT
		Done : BOOL;
		Status : UINT;
	END_VAR
	VAR
		intern : XSM_IO_Cfg_internType;
		AsIOAccWrite_0 : AsIOAccWrite;
		AsIOAccWriteReg_0 : AsIOAccWriteReg;
	END_VAR
END_FUNCTION_BLOCK

FUNCTION_BLOCK XSM_AcyclicRead (*Stepper motor acyclic reads.*)
	VAR_INPUT
		Enable : BOOL;
		Read : BOOL;
		Mode : USINT;
		Reset : BOOL;
		pIO_Mapping : UDINT;
	END_VAR
	VAR_OUTPUT
		ReadData : XSM_AcyclicReadDataType;
		Status : UINT;
	END_VAR
	VAR
		intern : XSM_AcyclicRead_internType;
		AsIOAccRead_0 : AsIOAccRead;
		AsIOAccReadReg_0 : AsIOAccReadReg;
	END_VAR
END_FUNCTION_BLOCK
```

#### XSM_Ramp.typ
```iecst
TYPE
	XSM_Ctrl_IOMappingType : 	STRUCT
		DeviceName : STRING[80];
		Channel : INT;
		ModuleOK : BOOL;
		ModuleID : UINT;
		AbsPos : DINT;
		MpGenControl : UINT;
		MpGenMode : SINT;
		AbsPosActVal : DINT;
		MpGenStatus : UINT;
		InputStatus : USINT;
	END_STRUCT;
	XSM_Ctrl_ParametersType : 	STRUCT
		Units_rev : UINT;
		PosSWLimit : DINT;
		NegSWLimit : DINT;
		HomePosition : DINT;
		HomeMode : USINT;
		Ignore_SWLimits : BOOL;
		Ignore_HWLimits : BOOL;
		HWLimits_Active_Low : BOOL;
		StallDetectionEnable : BOOL;
		UnderCurrentDetectionEnable : BOOL;
	END_STRUCT;
	XSM_IO_Cfg_internType : 	STRUCT
		StateMan : UINT;
		Cfg_State : USINT;
		OverflowWarning : DINT;
		AsIOAccWriteValue : REAL;
		ChannelName : STRING[30];
		Retries : USINT;
		IO_Mapping : XSM_Ctrl_IOMappingType;
		Parameters : XSM_Ctrl_ParametersType;
	END_STRUCT;
	XSM_IOCfg_CurrentType : 	STRUCT
		Holding : REAL;
		Rated : REAL;
		Maximum : REAL;
	END_STRUCT;
	XSM_IOCfg_StallType : 	STRUCT
		StallDetection : USINT;
		DisplayMotorLoadValues : BOOL;
	END_STRUCT;
	XSM_IOCfg_ReferencingType : 	STRUCT
		ReferencingConfiguration : SINT;
		StallRecongnitionDelay : USINT;
	END_STRUCT;
	XSM_IOCfg_MPGenType : 	STRUCT
		MaxSpeed : UINT;
		MaxAcc : UINT;
		MaxDec : UINT;
		RevLoop : INT;
		FixedPos_a : DINT;
		FixedPos_b : DINT;
		RefSpeed : DINT;
		JoltTimeLimitation : SINT;
	END_STRUCT;
	XSM_IO_ConfigurationType : 	STRUCT
		MixedDecayCfg : USINT;
		Current : XSM_IOCfg_CurrentType;
		FullStepThreshold : UINT;
		StallCfg : XSM_IOCfg_StallType;
		RefCfg : XSM_IOCfg_ReferencingType;
		MPGen : XSM_IOCfg_MPGenType;
	END_STRUCT;
	XSM_Ctrl_StateMachineType : 	STRUCT
		NotReadyToSwitchOn : BOOL;
		SwitchOnDisabled : BOOL;
		ReadyToSwitchOn : BOOL;
		SwitchedOn : BOOL;
		OperationEnabled : BOOL;
		QuickStopActive : BOOL;
		FaultReactionActive : BOOL;
		Fault : BOOL;
	END_STRUCT;
	XSM_Ctrl_internType : 	STRUCT
		StateMan : UINT;
		TaskCyclicTime : REAL;
		CyclicCounter : REAL;
		OldAbsPosActVal : DINT;
		Target : DINT;
		AbsPos : REAL;
		CmdHome : BOOL;
		CmdReset : BOOL;
		AutoReset : BOOL;
		CmdMove_Absolute : BOOL;
		CmdMove_Additive : BOOL;
		CmdMove_Velocity : BOOL;
		CmdMove_Adv_Two_Position_Mode : BOOL;
		CmdMove_Adv_FixedPos_a : BOOL;
		CmdMove_Adv_FixedPos_b : BOOL;
		CmdMove_Adv_Target_Mode : BOOL;
		OverflowWarning : UINT;
		ErrorCode : UINT;
		ChannelName : STRING[30];
		XSM_StateMachine : XSM_Ctrl_StateMachineType;
	END_STRUCT;
	XSM_Ctrl_AdvancedType : 	STRUCT
		Target_Mode : BOOL;
		Target_Position : DINT;
		Two_Position_Mode : BOOL;
		Move_FixedPos_a : BOOL;
		Move_FixedPos_b : BOOL;
	END_STRUCT;
	XSM_Ctrl_CmdType : 	STRUCT
		Move_Absolute : BOOL;
		Position : DINT;
		Move_Additive : BOOL;
		Distance : DINT;
		Move_Velocity : BOOL;
		Velocity : DINT;
		Stop : BOOL;
		Home : BOOL;
		Reset : BOOL;
		Advanced : XSM_Ctrl_AdvancedType;
	END_STRUCT;
	XSM_Ctrl_MonitorType : 	STRUCT
		Actual_Position : DINT;
		Actual_Velocity : DINT;
		StandStill : BOOL;
		Target_Reached : BOOL;
		Home_OK : BOOL;
		Input_1 : BOOL;
		Input_2 : BOOL;
		Input_3 : BOOL;
		Input_4 : BOOL;
	END_STRUCT;
	XSM_AcyclicReadDataType : 	STRUCT
		DC_BusVoltage : UINT;
		PowerStage_Temperature : SINT;
		Module_Temperature : SINT;
		Encoder_RefPosCyclicCounter : DINT;
		Encoder_ActualValue : DINT;
		Encoder_RefPosAcyclicCounter : DINT;
	END_STRUCT;
	XSM_AcyclicRead_internType : 	STRUCT
		StateMan : UINT;
		ChannelName : STRING[30];
		ReadOK : BOOL;
		Retries : USINT;
		IO_Mapping : XSM_Ctrl_IOMappingType;
	END_STRUCT;
END_TYPE
```

#### XSM_Ramp.var
```iecst
VAR CONSTANT
	XSM_CW_DISABLE_OPERATION : UINT := 7;
	XSM_CW_DISABLE_VOLTAGE : UINT := 0;
	XSM_CW_ENABLE_OPERATION : UINT := 15;
	XSM_CW_FAULT_RESET : UINT := 128;
	XSM_CW_QUICK_STOP : UINT := 2;
	XSM_CW_SHUTDOWN : UINT := 6;
	XSM_CW_SWITCH_ON : UINT := 7;
	XSM_MODE_HOME_NEGATIVE : SINT := -128;
	XSM_MODE_HOME_POSITIVE : SINT := -127;
	XSM_MODE_MOVE_FIXED_A : SINT := -125;
	XSM_MODE_MOVE_FIXED_B : SINT := -126;
	XSM_MODE_OFF : SINT := 0;
	XSM_MODE_POSITION : SINT := 1;
	XSM_MODE_SET_ACTUAL_POSITION : SINT := -122;
	XSM_MODE_SPEED : SINT := 2;
	XSM_MODE_TARGET : SINT := -123;
	XSM_MODE_TWO_POSITION : SINT := -124;
	XSM_RD_SM_FAULT : UINT := 16#0008;
	XSM_RD_SM_FAULT_REACTION_ACTIVE : UINT := 16#000F;
	XSM_RD_SM_NOT_READY_TO_SWITCH_ON : UINT := 16#0000;
	XSM_RD_SM_OPERATION_ENABLED : UINT := 16#0027;
	XSM_RD_SM_QUICK_STOP_ACTIVE : UINT := 16#0007;
	XSM_RD_SM_READY_TO_SWITCH_ON : UINT := 16#0021;
	XSM_RD_SM_SWITCH_ON_DISABLED : UINT := 16#0040;
	XSM_RD_SM_SWITCHED_ON : UINT := 16#0023;
	XSM_RD_STATE_MACHINE_MASK_ACTIVE : UINT := 16#006F;
	XSM_RD_STATE_MACHINE_MASK_STOP : UINT := 16#004F;
END_VAR
```
